// TIA Portal project "#06-J1500T(改角度）" (V17)

(* hardware
DEVICE "S7-1200 station_1"  S7-1200 Station
   slot 0: "Rack_0"  S7-1200 Rack  Rack  V1.0
   slot 1: "PLC_1"  CPU 1215C DC/DC/DC  6ES7 215-1AG40-0XB0  V4.5
   slot 2: "DI 16x24VDC_1"  6ES7 221-1BH32-0XB0  V2.0
   slot 3: "DI 16x24VDC_2"  6ES7 221-1BH32-0XB0  V2.0
   slot 4: "DI 16x24VDC_3"  6ES7 221-1BH32-0XB0  V2.0
   slot 5: "DQ 16x24VDC_1"  SM 1222 DQ16 x 24VDC  6ES7 222-1BH32-0XB0  V2.0
   slot 101: "CM 1243-5"  CM 1243-5  6GK7 243-5DX30-0XE0  V1.3
DEVICE "ET 200SP station_1"  ET 200SP-Station
   slot 0: "机架_0"  Rack  6ES5 710-8MAx1
   slot 0: "IO device_1"  IM 155-6 PN ST  6ES7 155-6AU01-0BN0  V4.2
   slot 1: "DI 16x24VDC ST_1"  DI 16x24VDC ST  6ES7 131-6BH01-0BA0  V0.0
      slot 1: "DI 16x24VDC ST_1"  DI 16x24VDC ST
   slot 2: "DI 16x24VDC ST_6"  DI 16x24VDC ST  6ES7 131-6BH01-0BA0  V0.0
      slot 1: "DI 16x24VDC ST_6"  DI 16x24VDC ST
   slot 3: "DI 16x24VDC ST_5"  DI 16x24VDC ST  6ES7 131-6BH01-0BA0  V0.0
      slot 1: "DI 16x24VDC ST_5"  DI 16x24VDC ST
   slot 4: "DI 16x24VDC ST_4"  DI 16x24VDC ST  6ES7 131-6BH01-0BA0  V0.0
      slot 1: "DI 16x24VDC ST_4"  DI 16x24VDC ST
   slot 5: "DI 16x24VDC ST_3"  DI 16x24VDC ST  6ES7 131-6BH01-0BA0  V0.0
      slot 1: "DI 16x24VDC ST_3"  DI 16x24VDC ST
   slot 6: "DQ 16x24VDC/0.5A ST_2"  DQ 16x24VDC/0.5A ST  6ES7 132-6BH01-0BA0  V0.0
      slot 1: "DQ 16x24VDC/0.5A ST_2"  DQ 16x24VDC/0.5A ST
   slot 7: "DQ 16x24VDC/0.5A ST_1"  DQ 16x24VDC/0.5A ST  6ES7 132-6BH01-0BA0  V0.0
      slot 1: "DQ 16x24VDC/0.5A ST_1"  DQ 16x24VDC/0.5A ST
   slot 8: "服务器模块_1"  Server module  6ES7 193-6PA00-0AA0  V1.1
      slot 1: "服务器模块_1"  Server module
   slot 127: "BA 2xRJ45"  BA 2xRJ45  6ES7 193-6AR00-0AA0  V0.0
      slot 1: "Port_1"  X1 P1 R  6ES7 193-6AR00-0AA0  V0.0
      slot 2: "Port_2"  X1 P2 R  6ES7 193-6AR00-0AA0  V0.0
DEVICE "HMI_1"  TP900 Comfort
   slot 0: "HMI_1"  TP900 Comfort  6AV2 124-0JC01-0AX0  15.1.0.0
   slot 1: "HMI_RT_1"  TP900 Comfort  6AV2 124-0JC01-0AX0  15.1.0.0
   slot 5: "HMI_1.IE_CP_1"  PROFINET Interface  15.0.1.0
      slot 1: "PROFINET Interface_1"  PROFINET Interface
         slot 1: "Port_1"  Port
         slot 2: "Port_2"  Port
   slot 7: "HMI_1.MPI/DP_CP_1"  MPI/DP Interface  15.0.1.0
DEVICE "GSD device_2"  GSD.Device
   slot 0: "机架_0"  Rail
   slot 0: "横梁站"  P+F  Encoder  4.0
DEVICE "GSD device_1"  GSD.Device
   slot 0: "机架_0"  Rail
   slot 0: "滑块站"  P+F  Encoder  4.0
*)

// ===== PLC "PLC_1"  CPU 1215C DC/DC/DC =====

VAR_GLOBAL   // PLC tag table "默认变量表"
   "Tag_1" AT %I0.0 : Bool;
   "Tag_136" AT %I19.3 : Bool;
   "Tag_137" AT %I19.4 : Bool;
   "Tag_138" AT %I19.5 : Bool;
   "Tag_139" AT %I19.6 : Bool;
   "Tag_140" AT %I19.7 : Bool;
   "机械凸轮单次返回" AT %I19.2 : Bool;
   "机械凸轮单次允许" AT %I19.1 : Bool;
   "机械凸轮上死点" AT %I19.0 : Bool;
   "右后双手闭点" AT %I18.7 : Bool;
   "Tag_46(1)" AT %I6.0 : Bool;
   "Tag_47(1)" AT %I6.1 : Bool;
   "Tag_48(1)" AT %I6.2 : Bool;
   "Tag_49(1)" AT %I6.3 : Bool;
   "Tag_50(1)" AT %I6.4 : Bool;
   "Tag_51(1)" AT %I6.5 : Bool;
   "Tag_52(1)" AT %I6.6 : Bool;
   "Tag_53(1)" AT %I6.7 : Bool;
   "Tag_54(1)" AT %I7.0 : Bool;
   "Tag_55(1)" AT %I7.1 : Bool;
   "Tag_56(1)" AT %I7.2 : Bool;
   "Tag_57(1)" AT %I7.3 : Bool;
   "Tag_58(1)" AT %I7.4 : Bool;
   "Tag_59" AT %I7.5 : Bool;
   "Tag_60" AT %I7.6 : Bool;
   "Tag_61(1)" AT %I7.7 : Bool;
   "工作台夹紧压检" AT %I18.0 : Bool;
   "工作台放松压检" AT %I18.1 : Bool;
   "故障复位" AT %I12.4 : Bool;
   "Tag_128" AT %I18.3 : Bool;
   "Tag_129" AT %I18.4 : Bool;
   "Tag_130" AT %I18.5 : Bool;
   "右后双手开点" AT %I18.6 : Bool;
   "Tag_108" AT %I15.7 : Bool;
   "平衡缸气压检测" AT %I15.6 : Bool;
   "Tag_105" AT %I15.4 : Bool;
   "Tag_28(1)" AT %I3.7 : Bool;
   "主电机启动接触器接通" AT %I3.5 : Bool;
   "Tag_26" AT %I3.4 : Bool;
   "Tag_25" AT %I3.3 : Bool;
   "Tag_2" AT %I0.1 : Bool;
   "Tag_3" AT %I0.2 : Bool;
   "Tag_4" AT %I0.3 : Bool;
   "Tag_5" AT %I0.4 : Bool;
   "Tag_6" AT %I0.5 : Bool;
   "Tag_7" AT %I0.6 : Bool;
   "Tag_8" AT %I0.7 : Bool;
   "Tag_9" AT %I1.0 : Bool;
   "Tag_10" AT %I1.1 : Bool;
   "Tag_11" AT %I1.2 : Bool;
   "Tag_12" AT %I1.3 : Bool;
   "Tag_13" AT %I1.4 : Bool;
   "Tag_14" AT %I1.5 : Bool;
   "Tag_15" AT %I2.1 : Bool;
   "Tag_16" AT %I2.2 : Bool;
   "Tag_17" AT %I2.3 : Bool;
   "KM17" AT %I2.4 : Bool;
   "Tag_19" AT %I2.5 : Bool;
   "Tag_20" AT %I2.6 : Bool;
   "Tag_21" AT %I2.7 : Bool;
   "KM12" AT %I3.0 : Bool;
   "Tag_23" AT %I3.1 : Bool;
   "KM11" AT %I3.2 : Bool;
   "Tag_35(1)" AT %I4.5 : Bool;
   "Tag_36(1)" AT %I4.6 : Bool;
   "Tag_37(1)" AT %I4.7 : Bool;
   "Tag_38(1)" AT %I5.0 : Bool;
   "Tag_39(1)" AT %I5.1 : Bool;
   "Tag_40(1)" AT %I5.2 : Bool;
   "Tag_41(1)" AT %I5.3 : Bool;
   "Tag_42(1)" AT %I5.4 : Bool;
   "Tag_43(1)" AT %I5.5 : Bool;
   "Tag_44(1)" AT %I5.6 : Bool;
   "Tag_45(1)" AT %I5.7 : Bool;
   "滑块调整选择" AT %I14.1 : Bool;
   "行程" AT %I14.2 : Bool;
   "气垫调整" AT %I14.3 : Bool;
   "模具更换" AT %I14.4 : Bool;
   "滑块向上" AT %I14.5 : Bool;
   "滑块向下" AT %I14.6 : Bool;
   "停上死点" AT %I14.7 : Bool;
   "Tag_101" AT %I15.0 : Bool;
   "滑块调整过扭矩" AT %I15.1 : Bool;
   "液压保护卸荷" AT %I15.2 : Bool;
   "液压保护压力检测" AT %I15.3 : Bool;
   "Tag_34(1)" AT %I4.4 : Bool;
   "爬梯开关" AT %I15.5 : Bool;
   "Tag_33(1)" AT %I4.3 : Bool;
   "Tag_31(1)" AT %I4.1 : Bool;
   "润滑停止按钮" AT %I10.0 : Bool;
   "润滑启动按钮" AT %I10.1 : Bool;
   "气垫手动润滑按钮" AT %I10.2 : Bool;
   "平衡缸手动润滑按钮" AT %I10.3 : Bool;
   "145" AT %I10.4 : Bool;
   "液压保护复位1" AT %I10.5 : Bool;
   "液压保护复位2" AT %I10.6 : Bool;
   "模具夹紧按钮" AT %I10.7 : Bool;
   "模具松开按钮" AT %I11.0 : Bool;
   "模具更换转换" AT %I11.1 : Bool;
   "工作台夹紧" AT %I11.2 : Bool;
   "工作台松开" AT %I11.3 : Bool;
   "微调启动按钮" AT %I11.4 : Bool;
   "微调正转" AT %I11.5 : Bool;
   "微调反转" AT %I11.6 : Bool;
   "主电机停止" AT %I11.7 : Bool;
   "Tag_30(1)" AT %I4.0 : Bool;
   "Tag_32(1)" AT %I4.2 : Bool;
   "Tag_61" AT %Q0.0 : Bool;
   "Tag_62" AT %Q0.1 : Bool;
   "Tag_63" AT %Q0.2 : Bool;
   "Tag_64" AT %Q0.3 : Bool;
   "Tag_65" AT %Q0.4 : Bool;
   "Tag_66" AT %Q0.5 : Bool;
   "Tag_68" AT %Q0.7 : Bool;
   "主电机正转DI1" AT %Q1.0 : Bool;
   "Tag_70" AT %Q1.1 : Bool;
   "润滑油泵启动2" AT %Q2.0 : Bool;
   "M6 ?" AT %Q2.1 : Bool;
   "KM3" AT %Q2.2 : Bool;
   "变频器上电" AT %Q2.3 : Bool;
   "气垫调整防粘连KM19" AT %Q2.4 : Bool;
   "气垫调整向上KM20" AT %Q2.5 : Bool;
   "气垫调整向下KM21" AT %Q2.6 : Bool;
   "Tag_67" AT %Q0.6 : Bool;
   "润滑油泵启动KM11" AT %Q2.7 : Bool;
   "滑块调整防粘连KM5" AT %Q3.0 : Bool;
   "滑块向上KM6" AT %Q3.1 : Bool;
   "滑块向下KM7" AT %Q3.2 : Bool;
   "制动器阀" AT %Q12.7 : Bool;
   "飞轮制动阀" AT %Q13.0 : Bool;
   "工作台夹紧阀(1)" AT %Q13.1 : Bool;
   "工作台放松阀(1)" AT %Q13.2 : Bool;
   "Tag_154" AT %Q13.3 : Bool;
   "Tag_155" AT %Q13.4 : Bool;
   "Tag_156" AT %Q13.5 : Bool;
   "Tag_157" AT %Q13.6 : Bool;
   "润滑指示灯" AT %Q13.7 : Bool;
   "下死点指示(1)" AT %Q10.0 : Bool;
   "离合器阀" AT %Q12.6 : Bool;
   "平衡缸润滑阀" AT %Q12.5 : Bool;
   "备用(4)" AT %Q12.3 : Bool;
   "KA41主电机正转" AT %Q3.3 : Bool;
   "Tag_83" AT %Q3.4 : Bool;
   "Tag_86" AT %Q3.5 : Bool;
   "Tag_87" AT %Q3.6 : Bool;
   "Tag_88" AT %Q3.7 : Bool;
   "上死点指示" AT %Q10.1 : Bool;
   "润滑油位低指示" AT %Q10.2 : Bool;
   "润滑油位高指示" AT %Q10.3 : Bool;
   "气垫润滑高压指示" AT %Q10.4 : Bool;
   "滤油器堵塞指示" AT %Q10.5 : Bool;
   "Tag_100" AT %Q10.6 : Bool;
   "Tag_102" AT %Q10.7 : Bool;
   "液压保护卸荷指示" AT %Q11.0 : Bool;
   "滑块调整过扭矩指示" AT %Q11.1 : Bool;
   "主电机运行指示" AT %Q11.2 : Bool;
   "连续预置指示" AT %Q11.3 : Bool;
   "Tag_109" AT %Q11.4 : Bool;
   "液压保护气源气阀(1)" AT %Q11.5 : Bool;
   "液压保护泵阀(1)" AT %Q11.6 : Bool;
   "Tag_142" AT %Q11.7 : Bool;
   "备用" AT %Q12.0 : Bool;
   "备用(1)" AT %Q12.1 : Bool;
   "备用(3)" AT %Q12.2 : Bool;
   "气垫润滑阀" AT %Q12.4 : Bool;
   "过滤器正常" AT %M5.0 : Bool;
   "润滑油压正常" AT %M5.1 : Bool;
   "滑块调整允许" AT %M5.2 : Bool;
   "急停故障" AT %M6.0 : Bool;
   "液压保护故障" AT %M6.1 : Bool;
   "气压故障" AT %M6.2 : Bool;
   "设备故障" AT %M6.3 : Bool;
   "滑块调整允许(1)" AT %M6.4 : Bool;
   "Tag_22" AT %MD20 : Time;
   "滑块调整允许2(1)" AT %M6.5 : Bool;
   "气垫调整允许" AT %M6.6 : Bool;
   "工作台移动允许" AT %M7.0 : Bool;
   "工作台落到位" AT %M7.1 : Bool;
   "润滑油泵启动OK" AT %M5.5 : Bool;
   "10度" AT %M200.0 : Bool;
   "20度" AT %M200.1 : Bool;
   "30度" AT %M200.2 : Bool;
   "40度" AT %M200.3 : Bool;
   "50" AT %M200.4 : Bool;
   "60" AT %M200.5 : Bool;
   "70" AT %M200.6 : Bool;
   "80" AT %M200.7 : Bool;
   "90" AT %M201.0 : Bool;
   "100" AT %M201.1 : Bool;
   "110" AT %M201.2 : Bool;
   "120" AT %M201.3 : Bool;
   "130" AT %M201.4 : Bool;
   "140" AT %M201.5 : Bool;
   "150" AT %M201.6 : Bool;
   "160" AT %M201.7 : Bool;
   "170" AT %M202.0 : Bool;
   "180" AT %M202.1 : Bool;
   "190" AT %M202.2 : Bool;
   "200" AT %M202.3 : Bool;
   "210" AT %M202.4 : Bool;
   "220" AT %M202.5 : Bool;
   "230" AT %M202.6 : Bool;
   "240" AT %M202.7 : Bool;
   "250" AT %M203.0 : Bool;
   "260" AT %M203.1 : Bool;
   "270" AT %M203.2 : Bool;
   "280" AT %M203.3 : Bool;
   "290" AT %M203.4 : Bool;
   "300" AT %M203.5 : Bool;
   "310" AT %M203.6 : Bool;
   "320" AT %M203.7 : Bool;
   "330" AT %M204.0 : Bool;
   "340" AT %M204.1 : Bool;
   "350" AT %M204.2 : Bool;
   "360" AT %M204.3 : Bool;
   "上死点" AT %M204.4 : Bool;
   "制动监控" AT %M204.5 : Bool;
   "下死点" AT %M204.6 : Bool;
   "单次返回" AT %M204.7 : Bool;
   "光电保护位置" AT %M205.0 : Bool;
   "横梁编码器" AT %ID68 : DWord;
   "滑块编码器" AT %ID72 : DInt;
   "主电机启动1" AT %I12.0 : Bool;
   "微调选择(1)" AT %I14.0 : Bool;
   "主电机启动2" AT %I12.1 : Bool;
   "寸动开点1" AT %I12.2 : Bool;
   "寸动闭点1" AT %I12.3 : Bool;
   "故障复位(1)" AT %I18.2 : Bool;
   "寸动开点2" AT %I12.5 : Bool;
   "寸动闭点2" AT %I12.6 : Bool;
   "Tag_34" AT %I12.7 : Bool;
   "Tag_35" AT %I13.0 : Bool;
   "选择连续" AT %I13.1 : Bool;
   "单次选择" AT %I13.2 : Bool;
   "选择寸动" AT %I13.3 : Bool;
   "Tag_39" AT %I13.4 : Bool;
   "急停闭点" AT %I13.5 : Bool;
   "急停开点1" AT %I13.6 : Bool;
   "急停开点2" AT %I13.7 : Bool;
   "润滑油位高" AT %I16.0 : Bool;
   "润滑油位低" AT %I16.1 : Bool;
   "Tag_45" AT %I16.2 : Bool;
   "润滑低压1" AT %I16.3 : Bool;
   "润滑低压2" AT %I16.4 : Bool;
   "润滑低压3" AT %I16.5 : Bool;
   "润滑高压" AT %I16.6 : Bool;
   "滤油器堵塞1" AT %I16.7 : Bool;
   "滤油器堵塞2" AT %I17.0 : Bool;
   "滤油器堵塞3" AT %I17.1 : Bool;
   "Tag_53" AT %I17.2 : Bool;
   "工作台落到位前" AT %I17.3 : Bool;
   "工作台落到位后" AT %I17.4 : Bool;
   "气垫落到位" AT %I17.5 : Bool;
   "右前双手开点" AT %I17.6 : Bool;
   "右前双手闭点" AT %I17.7 : Bool;
   "急停正常" AT %M10.0 : Bool;
   "行程允许" AT %M14.0 : Bool;
   "寸动允许" AT %M14.1 : Bool;
   "寸动开始" AT %M14.2 : Bool;
   "单次允许" AT %M14.3 : Bool;
   "单次开始" AT %M14.4 : Bool;
   "双手按钮开点" AT %M14.5 : Bool;
   "双手按钮闭点" AT %M14.6 : Bool;
   "编码器闭点监控" AT %M14.7 : Bool;
   "编码器开点监控" AT %M15.0 : Bool;
   "编码器故障" AT %M15.1 : Bool;
   "工作台-夹紧OK" AT %M15.2 : Bool;
   "工作台放松OK" AT %M15.3 : Bool;
   "润滑正常" AT %M15.4 : Bool;
   "滑块软限位上" AT %M15.5 : Bool;
   "滑块软限位下" AT %M15.6 : Bool;
   "上调整设定值" AT %M15.7 : Bool;
   "滑块调整自动向上" AT %M16.0 : Bool;
   "滑块调整自动向下" AT %M16.1 : Bool;
   "滑块调整自动选择" AT %M16.2 : Bool;
   "滑块手动调整" AT %M16.3 : Bool;
   "滑块调整手动/自动" AT %M301.5 : Bool;
   "ECamdata _DB_D{10}滑块设定高度" AT %MD150 : Real;
   "润滑检测时间" AT %M600.0 : Bool;
   "气垫向上调整" AT %M220.0 : Bool;
   "气垫向下调整" AT %M220.1 : Bool;
   "System_Byte" AT %MB1 : Byte;
   "FirstScan" AT %M1.0 : Bool;
   "DiagStatusUpdate" AT %M1.1 : Bool;
   "AlwaysTRUE" AT %M1.2 : Bool;
   "AlwaysFALSE" AT %M1.3 : Bool;
   "Clock_Byte" AT %MB0 : Byte;
   "Clock_10Hz" AT %M0.0 : Bool;
   "Clock_5Hz" AT %M0.1 : Bool;
   "Clock_2.5Hz" AT %M0.2 : Bool;
   "Clock_2Hz" AT %M0.3 : Bool;
   "Clock_1.25Hz" AT %M0.4 : Bool;
   "Clock_1Hz" AT %M0.5 : Bool;
   "Clock_0.625Hz" AT %M0.6 : Bool;
   "Clock_0.5Hz" AT %M0.7 : Bool;
   "主电机启动标志" AT %M700.0 : Bool;
   "爬梯占位" AT %M5000.1 : Bool;
   "正传选择（占位）" AT %M5000.2 : Bool;
   "反转选择（占位）" AT %M5000.3 : Bool;
   "正转启动标志" AT %M700.1 : Bool;
   "反转启动标志" AT %M700.2 : Bool;
   "主电机反转（占位）" AT %M5000.4 : Bool;
   "主电机转速稳定" AT %M700.3 : Bool;
   "横梁编码器通讯故障" AT %M700.5 : Bool;
   "滑块编码器通讯故障" AT %M700.6 : Bool;
   "ET200通讯故障" AT %M700.7 : Bool;
   "单次允许1" AT %M205.2 : Bool;
   "Tag_18" AT %M19.2 : Bool;
   "防重复角度" AT %M205.1 : Bool;
   "防重复监控" AT %M702.0 : Bool;
   "单次条件3" AT %M18.1 : Bool;
   "临时屏蔽" AT %M1000.0 : Bool;
END_VAR

VAR_GLOBAL   // PLC tag table "变量表"
   "平衡缸压力模拟量" AT %ID80 : DWord;
   "气垫压力模拟量" AT %ID81 : DWord;
   "Tag_108(1)" AT %QW570 : Int;
   "Tag_109(1)" AT %QW572 : Int;
   "报警1" AT %M3000.0 : Bool;
   "报警2" AT %M3000.1 : Bool;
   "报警3" AT %M3000.2 : Bool;
   "报警4" AT %M3000.3 : Bool;
   "报警5" AT %M3000.4 : Bool;
   "报警6" AT %M3000.5 : Bool;
   "报警7" AT %M3000.6 : Bool;
   "报警8" AT %M3000.7 : Bool;
   "报警9" AT %M3001.0 : Bool;
   "报警10" AT %M3001.1 : Bool;
   "报警11" AT %M3001.2 : Bool;
   "报警12" AT %M3001.3 : Bool;
   "报警13" AT %M3001.4 : Bool;
   "报警14" AT %M3001.5 : Bool;
   "报警15" AT %M3001.6 : Bool;
   "报警16" AT %M3001.7 : Bool;
   "PLC报警变量组1" AT %MW3000 : Int;
   "PLC报警变量组2" AT %MW3002 : Int;
   "PLC报警变量组3" AT %MW3004 : Int;
   "报警17" AT %M3002.0 : Bool;
   "报警18" AT %M3002.1 : Bool;
   "报警19" AT %M3002.2 : Bool;
   "报警20" AT %M3002.3 : Bool;
   "报警21" AT %M3002.4 : Bool;
   "报警22" AT %M3002.5 : Bool;
   "报警23" AT %M3002.6 : Bool;
   "报警24" AT %M3002.7 : Bool;
   "报警25" AT %M3003.0 : Bool;
   "报警26" AT %M3003.1 : Bool;
   "报警27" AT %M3003.2 : Bool;
   "报警28" AT %M3003.3 : Bool;
   "报警29" AT %M3003.4 : Bool;
   "报警30" AT %M3003.5 : Bool;
   "报警31" AT %M3003.6 : Bool;
   "报警32" AT %M3003.7 : Bool;
   "报警33" AT %M3004.0 : Bool;
   "报警34" AT %M3004.1 : Bool;
   "报警35" AT %M3004.2 : Bool;
   "报警36" AT %M3004.3 : Bool;
   "报警37" AT %M3004.4 : Bool;
   "报警38" AT %M3004.5 : Bool;
   "报警39" AT %M3004.6 : Bool;
   "报警40" AT %M3004.7 : Bool;
   "报警41" AT %M3005.0 : Bool;
   "报警42" AT %M3005.1 : Bool;
   "报警43" AT %M3005.2 : Bool;
   "报警44" AT %M3005.3 : Bool;
   "报警45" AT %M3005.4 : Bool;
   "报警46" AT %M3005.5 : Bool;
   "报警47" AT %M3005.6 : Bool;
   "报警48" AT %M3005.7 : Bool;
   "Tag_1(1)" AT %M100.0 : Bool;
   "Tag_7(2)" AT %M100.1 : Bool;
   "异常报警1" AT %M1008.3 : Bool;
   "异常报警2" AT %M1008.4 : Bool;
   "计数开始" AT %M30.0 : Bool;
   "计数清零" AT %M30.1 : Bool;
   "产量到达" AT %M30.2 : Bool;
END_VAR

VAR_GLOBAL CONSTANT   // PLC tag table "变量表"
   "无(1)" : Pip := 65535;
   "自动更新(1)" : Pip := 0;
   "PIP 1(1)" : Pip := 1;
   "PIP 2(1)" : Pip := 2;
   "PIP 3(1)" : Pip := 3;
   "PIP 4(1)" : Pip := 4;
   "PIP OB 伺服(1)" : Pip := 32768;
   "Local~MC(1)" : Hw_SubModule := 51;
   "Local~Common(1)" : Hw_SubModule := 50;
   "Local~Device(1)" : Hw_Device := 32;
   "Local~Configuration(1)" : Hw_SubModule := 33;
   "Local~Exec(1)" : Hw_SubModule := 52;
   "Local(1)" : Hw_SubModule := 49;
   "Local~PROFINET_接口_1(1)" : Hw_Interface := 64;
   "Local~PROFINET_接口_1~端口_1(1)" : Hw_Interface := 65;
   "Local~HSC_1(1)" : Hw_Hsc := 257;
   "Local~HSC_2(1)" : Hw_Hsc := 258;
   "Local~HSC_3(1)" : Hw_Hsc := 259;
   "Local~HSC_4(1)" : Hw_Hsc := 260;
   "Local~HSC_5(1)" : Hw_Hsc := 261;
   "Local~HSC_6(1)" : Hw_Hsc := 262;
   "Local~AI_2_1" : Hw_SubModule := 263;
   "Local~DI_14_DQ_10_1(1)" : Hw_SubModule := 264;
   "Local~Pulse_1(1)" : Hw_Pwm := 265;
   "Local~Pulse_2(1)" : Hw_Pwm := 266;
   "Local~Pulse_3(1)" : Hw_Pwm := 267;
   "Local~Pulse_4(1)" : Hw_Pwm := 268;
   "Local~CM_1243-5~DP_接口(1)" : Hw_Interface := 269;
   "Local~CM_1243-5(1)" : Hw_SubModule := 271;
   "Local~PROFINET_IO-System(1)" : Hw_IoSystem := 272;
   "Local~DP-Mastersystem(1)" : Hw_IoSystem := 273;
   "Local~DI_16x24VDC_1(1)" : Hw_SubModule := 291;
   "Local~DI_16x24VDC_2(1)" : Hw_SubModule := 292;
   "Local~DQ_16x24VDC_1(1)" : Hw_SubModule := 293;
   "立柱右前操作站~Head" : Hw_Interface := 288;
   "立柱右前操作站~DPSlave" : Hw_DpSlave := 286;
   "立柱右前操作站~DI_32x24VDC_1" : Hw_SubModule := 289;
   "立柱右前操作站~AI_8x12BIT_1" : Hw_SubModule := 294;
   "立柱右前操作站~DI_32x24VDC_2" : Hw_SubModule := 295;
   "立柱右前操作站~DI_32x24VDC_3" : Hw_SubModule := 296;
   "立柱右前操作站~DI_32x24VDC_4" : Hw_SubModule := 297;
   "立柱右前操作站~DO_32x24VDC_0_5A_2" : Hw_SubModule := 299;
   "立柱右前操作站~DO_16x24VDC_0_5A_1" : Hw_SubModule := 290;
   "立柱右前操作站~DI_16x24VDC_1" : Hw_SubModule := 274;
   "横梁站~Head(1)" : Hw_Interface := 280;
   "横梁站~DPSlave(1)" : Hw_DpSlave := 278;
   "横梁站~P+F_Version_2_1_Singleturn_1(1)" : Hw_SubModule := 281;
   "OB_Main(1)" : OB_PCYCLE := 1;
   "OB_Cyclic interrupt" : OB_Cyclic := 30;
   "OB_RackStationFailure" : OB_Any := 86;
   "OB_Startup" : OB_STARTUP := 100;
   "滑块站~Head(1)" : Hw_Interface := 277;
   "滑块站~DPSlave(1)" : Hw_DpSlave := 275;
   "滑块站~32_Bit_Class_2_+_Speed_2_1" : Hw_SubModule := 282;
   "滑块站~32_Bit_Class_2_+_Speed_2_2" : Hw_SubModule := 283;
END_VAR

TYPE "用户数据类型_1"
   STRUCT
      Element_1 : Bool;
   END_STRUCT;
END_TYPE

// folder: 4.1_Line_Operation

TYPE "Operation_Mode"
   STRUCT
      Auto : Bool;
      Auto_Sim : Bool;
      APC : Bool;
      ATC : Bool;
      Man : Bool;
      Setup : Bool;
      工作模式 : UInt;
      零件表 : UInt;
   END_STRUCT;
END_TYPE

TYPE "4.1_Line_Operation"
   STRUCT
      Mode_Act : "Operation_Mode";
      Mode_Seting : "Operation_Mode";
      Recipes_Operation : "HMI_Recipe";
      HMI : Array[1..10] of "HMI_State";
   END_STRUCT;
END_TYPE

TYPE "HMI_Recipe"
   STRUCT
      Recipe : Struct
         Clear : Bool;
         Load : Bool;
         Save : Bool;
         Edit_No : Int;
         Recipe_Edit_Auth : Bool;
         Recipe_Edit_Wizard : Int;
         Load_Active : Bool;
         Save_Active : Bool;
         ii : Int;
         Load_Timer : IEC_TIMER;
         Save_Timer : IEC_TIMER;
      END_STRUCT;
      RecipeExport : Struct
         Done : Bool;
         Busy : Bool;
         Error : Bool;
         Status : Word;
      END_STRUCT;
      RecipeImport : Struct
         Done : Bool;
         Busy : Bool;
         Error : Bool;
         Status : Word;
      END_STRUCT;
   END_STRUCT;
END_TYPE

TYPE "HMI_State"
   STRUCT
      Command : Struct
         Doub_Part_Dropped_Mem : Bool;
         Part_Dropped_Mem : Bool;
         Part_Picker_Mem : Bool;
         Part_Done_Mem : Bool;
         Optim_Auth : Bool;
         Part_No_Chg_Auth : Bool;
      END_STRUCT;
      State : Struct
         Doub_Part_Dropped_Mem_1 : Bool;
         Part_Dropped_Mem_1 : Bool;
         Part_Picker_Mem_1 : Bool;
         Part_Done_Mem_1 : Bool;
      END_STRUCT;
   END_STRUCT;
END_TYPE

// folder: (top level)

DATA_BLOCK "中继"   // DB1
{ S7_Optimized_Access := 'TRUE' }
VERSION : 0.1
   VAR
      计数开关 : Bool;
      计数清零开关 : Bool;
      产量到达 : Bool;
   END_VAR
BEGIN
END_DATA_BLOCK

DATA_BLOCK "横梁编码器 _DB"   // DB3
{ S7_Optimized_Access := 'TRUE' }
VERSION : 0.1
   VAR
      "0.0" : Struct
         "+0.0" : DWord;
         "+4.0" : DWord;
         "+8.0" : DWord;
         "+12.0" : DWord;
      END_STRUCT;
      横梁 : Int;
      滑块 : Int;
      滑块_1 : DWord;
      "+0.3" : Int;
      "+0.4" : Int;
      "+0.5" : Int;
      "角度校准值(原+0.6）" : Int;
      编码器角度 : Int;
      "+0.7" : Int;
   END_VAR
   VAR RETAIN
      "+0.8" : Int;
   END_VAR
   VAR
      "+0.9" : Int;
      "+0.10" : Int;
      "0.11" : Real;
      平衡器分油器检测 : Int;
      横梁分油器检测 : Int;
      滑块分油器检测 : Int;
      气垫分油器检测 : Int;
      "+0.15" : Int;
      "+0.16" : Int;
      "+0.17" : Int;
      "+0.18" : Int;
      "+0.19" : Int;
      "+0.20" : Int;
      "+0.21" : Int;
      "+0.22" : Int;
      "+0.23" : Int;
      "+0.24" : Int;
      "+0.25" : Int;
      "+0.26" : Int;
      "+0.27" : Int;
      "+0.28" : Int;
      "+0.29" : Int;
      "+0.30" : Int;
      平衡器打油次数 : Int;
      主分油器打油次数 : Int;
      滑块打油次数 : Int;
      气点垫打油次数 : Int;
      "+0.35" : Int;
      "+0.36" : Int;
      "+0.37" : Int;
      "+0.38" : Int;
      "+0.39" : Int;
      "+0.40" : Int;
      "+0.41" : Int;
      "+0.42" : Int;
      "+0.43" : Int;
      "+0.44" : Int;
      "+0.45" : Int;
      "+0.46" : Int;
      "+0.47" : Int;
      "+0.48" : Int;
   END_VAR
   VAR RETAIN
      AI : Array[0..10] of DInt;
      D : Array[0..10] of Real;
   END_VAR
   VAR
      AQD : Real;
      产量设定 : Int;
      D107 : Real;
   END_VAR
BEGIN
END_DATA_BLOCK

DATA_BLOCK "数据块_2"   // DB6
{ S7_Optimized_Access := 'TRUE' }
VERSION : 0.1
BEGIN
END_DATA_BLOCK

DATA_BLOCK "ECamdata _DB"   // DB7
{ S7_Optimized_Access := 'TRUE' }
VERSION : 0.1
   VAR
      "0.0" : Struct
         "+0.0" : DWord;
         "+4.0" : DWord;
         "+8.0" : DWord;
         "+12.0" : DWord;
      END_STRUCT;
      横梁编码器 : Int;
      滑块编码器 : DInt;
      气垫编码器1 : DWord;
      气垫编码器2 : DWord;
      平衡器压力显示_3 : Int;
      电子凸轮编码器 : Int;
      "+0.5" : Real;
      电子凸轮编码器显示 : Int;
      "+0.7" : DInt;
      "+0.8" : Int;
      "+0.9" : Real;
      "+0.10_1" : Int;
      "+0.11" : Int;
      "+0.12" : Int;
      "+0.13" : Int;
      "+0.10" : Int;
      平衡器分油器检测 : Int;
      横梁分油器检测 : Int;
      滑块分油器检测 : Int;
      气垫分油器检测 : Int;
      "+0.15" : Int;
      "+0.16" : Int;
      "+0.17" : Int;
      "+0.18" : Int;
      "+0.19" : Int;
      "+0.20" : Int;
      "+0.21" : Int;
      "+0.22" : Int;
      "+0.23" : Int;
      "+0.24" : Int;
      "+0.25" : Int;
      "+0.26" : Int;
      "+0.27" : Int;
      "+0.28" : Int;
      "+0.29" : Int;
      "+0.30" : Int;
      平衡器打油次数 : Int;
      主分油器打油次数 : Int;
      滑块打油次数 : Int;
      气点垫打油次数 : Int;
      "+0.35" : Int;
      "+0.36" : Int;
      平衡器压力显示_2 : Real;
      平衡器压力显示_1 : Real;
      "+0.39" : Int;
      "+0.40" : Real;
      "+0.41" : Real;
      气垫模拟量 : Int;
      气垫模拟量_1 : Real;
      气垫模拟量_2 : Real;
      "+0.45" : DInt;
      "+0.46" : Int;
      "+0.47" : Real;
      "+0.48" : Int;
   END_VAR
   VAR RETAIN
      AI : Array[0..10] of DInt;
      D : Array[0..20] of Real;
   END_VAR
   VAR
      平衡器压力显示 : Real;
      AQD2 : Real;
      气垫模拟量显示1 : Real;
      气垫模拟量显示2 : Real;
      平衡器设置压力 : Real;
      气垫1压力设置 : Real;
      气垫2压力设置 : Real;
      D100 : Real;
      D101 : Int;
      D102 : Int;
      D103 : Real;
      D104 : Real;
      D105 : Real;
      D106 : Real;
      D107 : Int;
      D108 : Real;
      D109 : Real;
   END_VAR
   VAR RETAIN
      设置产量 : Int;
      当前产量 : Int;
      滑块位置 : Int;
   END_VAR
   VAR
      气垫位置 : Int;
   END_VAR
   VAR RETAIN
      D200 : DInt;
      D201 : Int;
   END_VAR
   VAR
      滑块中间值1 : Real;
   END_VAR
BEGIN
END_DATA_BLOCK

DATA_BLOCK "诊断数据"   // DB20
{ S7_Optimized_Access := 'TRUE' }
VERSION : 0.1
   VAR
      "横梁编码器-state" : Array[0..127] of Bool;
      "横梁编码器-return" : Word;
      "滑块编码器-state" : Array[0..127] of Bool;
      "滑块编码器-return" : Word;
      "ET200-state" : Array[0..127] of Bool;
      "ET200-return" : Word;
   END_VAR
BEGIN
END_DATA_BLOCK

DATA_BLOCK "中间变量"   // DB100
{ S7_Optimized_Access := 'TRUE' }
VERSION : 0.1
   VAR
      当前产量 : Int;
      目标产量 : Int;
   END_VAR
BEGIN
END_DATA_BLOCK

DATA_BLOCK "counter"   // DB101
{ S7_Optimized_Access := 'TRUE' }
VERSION : 0.1
   VAR
      产量计数 : IEC_COUNTER;
   END_VAR
BEGIN
END_DATA_BLOCK

DATA_BLOCK "timer"   // DB200
{ S7_Optimized_Access := 'TRUE' }
VERSION : 0.1
   VAR
      主电机转速稳定延时 : IEC_TIMER;
      清零防误触延时 : IEC_TIMER;
   END_VAR
BEGIN
END_DATA_BLOCK

// folder: 04_HMI_Comand_Config

DATA_BLOCK "Line_OP"   // DB10
{ S7_Optimized_Access := 'TRUE' }
VERSION : 0.1
BEGIN
END_DATA_BLOCK

// folder: System blocks/Program resources

DATA_BLOCK "IEC_Timer_0_DB_3"   // DB2
{ S7_Optimized_Access := 'TRUE' }
AUTHOR : Simatic
FAMILY : IEC
NAME : IEC_TMR
VERSION : 1.0
// stored: InstanceOfName IEC_TIMER
"IEC_TIMER"
BEGIN
END_DATA_BLOCK

DATA_BLOCK "IEC_Timer_0_DB_1"   // DB4
{ S7_Optimized_Access := 'TRUE' }
AUTHOR : Simatic
FAMILY : IEC
NAME : IEC_TMR
VERSION : 1.0
// stored: InstanceOfName IEC_TIMER
"IEC_TIMER"
BEGIN
END_DATA_BLOCK

DATA_BLOCK "IEC_Timer_0_DB_2"   // DB5
{ S7_Optimized_Access := 'TRUE' }
AUTHOR : Simatic
FAMILY : IEC
NAME : IEC_TMR
VERSION : 1.0
// stored: InstanceOfName IEC_TIMER
"IEC_TIMER"
BEGIN
END_DATA_BLOCK

DATA_BLOCK "当前产量"   // DB8
{ S7_Optimized_Access := 'TRUE' }
AUTHOR : Simatic
FAMILY : IEC
NAME : CNTR
VERSION : 1.0
// stored: InstanceOfName IEC_COUNTER
"IEC_COUNTER"
BEGIN
END_DATA_BLOCK

// folder: (top level)

FUNCTION "工作台移动" : Void   // FC1, LAD
{ S7_Optimized_Access := 'TRUE' }
VERSION : 0.1
BEGIN

REGION Network 2
   // 000000000000000000000000000000000000.
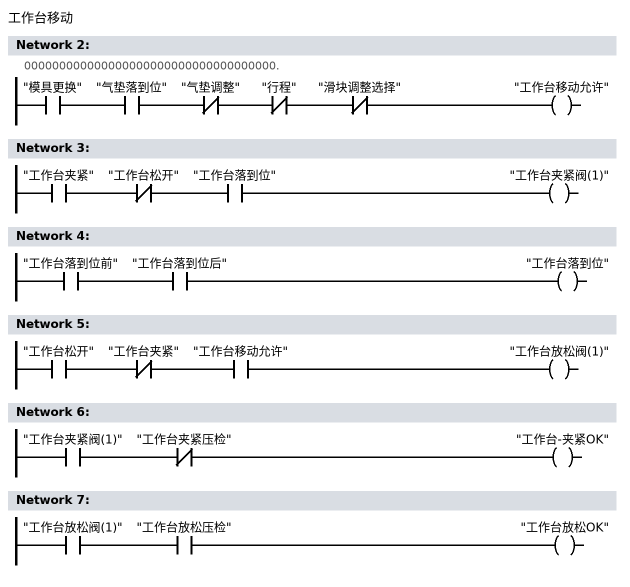
   RUNG wire#powerrail
      Contact( "模具更换" )
      Contact( "气垫落到位" )
      I_Contact( "气垫调整" )
      I_Contact( "行程" )
      I_Contact( "滑块调整选择" )
      Coil( "工作台移动允许" )
   END_RUNG
   // the same network as SCL:
   "工作台移动允许" := "模具更换" AND "气垫落到位" AND NOT "气垫调整" AND NOT "行程" AND NOT "滑块调整选择";
END_REGION

REGION Network 3
   RUNG wire#powerrail
      Contact( "工作台夹紧" )
      I_Contact( "工作台松开" )
      Contact( "工作台落到位" )
      Coil( "工作台夹紧阀(1)" )
   END_RUNG
   // the same network as SCL:
   "工作台夹紧阀(1)" := "工作台夹紧" AND NOT "工作台松开" AND "工作台落到位";
END_REGION

REGION Network 4
   RUNG wire#powerrail
      Contact( "工作台落到位前" )
      Contact( "工作台落到位后" )
      Coil( "工作台落到位" )
   END_RUNG
   // the same network as SCL:
   "工作台落到位" := "工作台落到位前" AND "工作台落到位后";
END_REGION

REGION Network 5
   RUNG wire#powerrail
      Contact( "工作台松开" )
      I_Contact( "工作台夹紧" )
      Contact( "工作台移动允许" )
      Coil( "工作台放松阀(1)" )
   END_RUNG
   // the same network as SCL:
   "工作台放松阀(1)" := "工作台松开" AND NOT "工作台夹紧" AND "工作台移动允许";
END_REGION

REGION Network 6
   RUNG wire#powerrail
      Contact( "工作台夹紧阀(1)" )
      I_Contact( "工作台夹紧压检" )
      Coil( "工作台-夹紧OK" )
   END_RUNG
   // the same network as SCL:
   "工作台-夹紧OK" := "工作台夹紧阀(1)" AND NOT "工作台夹紧压检";
END_REGION

REGION Network 7
   RUNG wire#powerrail
      Contact( "工作台放松阀(1)" )
      Contact( "工作台放松压检" )
      Coil( "工作台放松OK" )
   END_RUNG
   // the same network as SCL:
   "工作台放松OK" := "工作台放松阀(1)" AND "工作台放松压检";
END_REGION
END_FUNCTION

FUNCTION "横梁编码器调制" : Void   // FC2, LAD
{ S7_Optimized_Access := 'TRUE' }
VERSION : 0.1
BEGIN

REGION Network 1
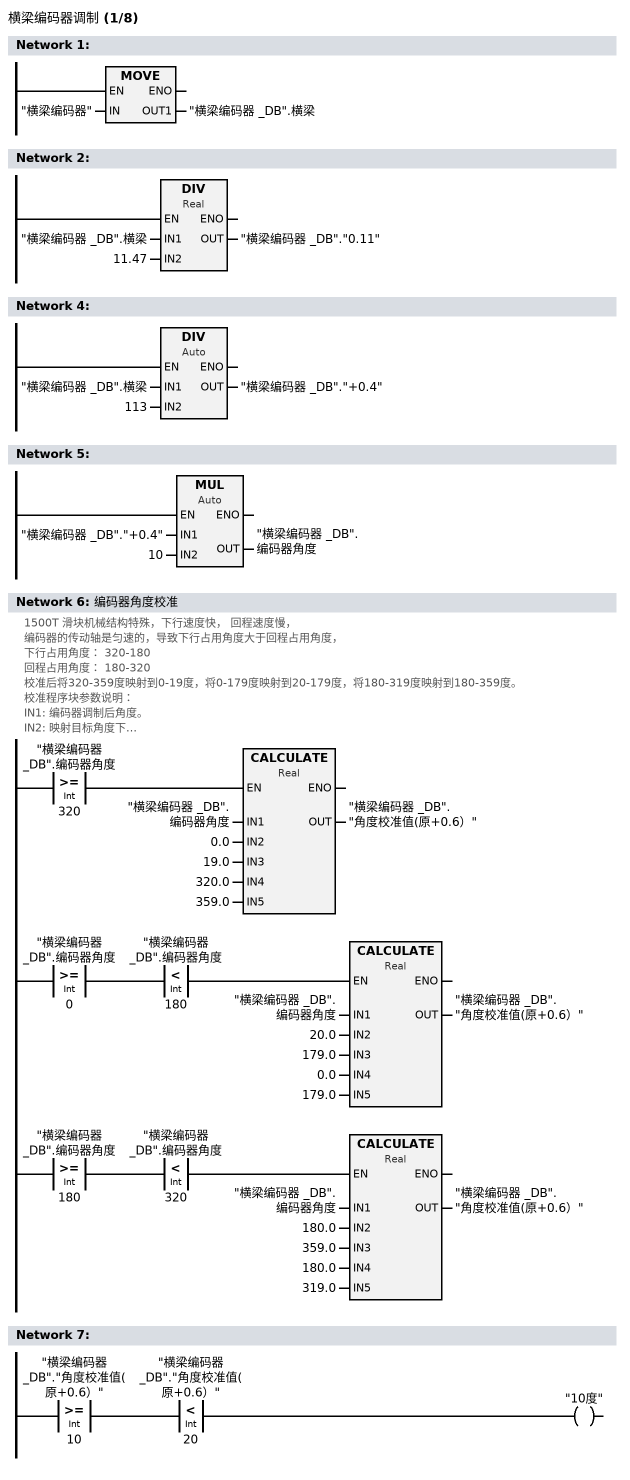
   RUNG wire#powerrail
      Move(in := "横梁编码器", out1 => "横梁编码器 _DB".横梁)
   END_RUNG
   // the same network as SCL:
   "横梁编码器 _DB".横梁 := "横梁编码器";
END_REGION

REGION Network 2
   RUNG wire#powerrail
      { S7_Templates := "SrcType := Real" } Div(in1 := "横梁编码器 _DB".横梁, in2 := 11.47, out => "横梁编码器 _DB"."0.11")
   END_RUNG
   // the same network as SCL:
   "横梁编码器 _DB"."0.11" := "横梁编码器 _DB".横梁 / 11.47;
END_REGION

REGION Network 4
   RUNG wire#powerrail
      Div(in1 := "横梁编码器 _DB".横梁, in2 := 113, out => "横梁编码器 _DB"."+0.4")
   END_RUNG
   // the same network as SCL:
   "横梁编码器 _DB"."+0.4" := "横梁编码器 _DB".横梁 / 113;
END_REGION

REGION Network 5
   RUNG wire#powerrail
      Mul(in1 := "横梁编码器 _DB"."+0.4", in2 := 10, out => "横梁编码器 _DB".编码器角度)
   END_RUNG
   // the same network as SCL:
   "横梁编码器 _DB".编码器角度 := "横梁编码器 _DB"."+0.4" * 10;
END_REGION

REGION Network 6: 编码器角度校准
   // 1500T 滑块机械结构特殊，下行速度快， 回程速度慢， 编码器的传动轴是匀速的，导致下行占用角度大于回程占用角度，
   // 下行占用角度： 320-180
   // 回程占用角度： 180-320
   // 校准后将320-359度映射到0-19度，将0-179度映射到20-179度，将180-319度映射到180-359度。 
   // 
   // 校准程序块参数说明： 
   // IN1: 编码器调制后角度。
   // IN2: 映射目标角度下限
   // IN3: 映射目标角度上限
   // IN4: 被映射角度下限
   // IN4: 被映射角度上限
   // OUT: 映射校准后的滑块实际角度
   RUNG wire#powerrail
      { S7_Templates := "SrcType := Int" } GE_Contact(in1 := "横梁编码器 _DB".编码器角度, in2 := 320)
      { S7_Templates := "SrcType := Real"; S7_Expression := "(IN1-IN4)/(IN5-IN4)*(IN3-IN2)+IN2" } Calculate(in1 := "横梁编码器 _DB".编码器角度, in2 := 0.0, in3 := 19.0, in4 := 320.0, in5 := 359.0, out => "横梁编码器 _DB"."角度校准值(原+0.6）")
   END_RUNG
   RUNG wire#powerrail
      { S7_Templates := "SrcType := Int" } GE_Contact(in1 := "横梁编码器 _DB".编码器角度, in2 := 0)
      { S7_Templates := "SrcType := Int" } LT_Contact(in1 := "横梁编码器 _DB".编码器角度, in2 := 180)
      { S7_Templates := "SrcType := Real"; S7_Expression := "(IN1-IN4)/(IN5-IN4)*(IN3-IN2)+IN2" } Calculate(in1 := "横梁编码器 _DB".编码器角度, in2 := 20.0, in3 := 179.0, in4 := 0.0, in5 := 179.0, out => "横梁编码器 _DB"."角度校准值(原+0.6）")
   END_RUNG
   RUNG wire#powerrail
      { S7_Templates := "SrcType := Int" } GE_Contact(in1 := "横梁编码器 _DB".编码器角度, in2 := 180)
      { S7_Templates := "SrcType := Int" } LT_Contact(in1 := "横梁编码器 _DB".编码器角度, in2 := 320)
      { S7_Templates := "SrcType := Real"; S7_Expression := "(IN1-IN4)/(IN5-IN4)*(IN3-IN2)+IN2" } Calculate(in1 := "横梁编码器 _DB".编码器角度, in2 := 180.0, in3 := 359.0, in4 := 180.0, in5 := 319.0, out => "横梁编码器 _DB"."角度校准值(原+0.6）")
   END_RUNG
   // the same network as SCL:
   IF "横梁编码器 _DB".编码器角度 >= 320 THEN
       "横梁编码器 _DB"."角度校准值(原+0.6）" := ("横梁编码器 _DB".编码器角度-320.0)/(359.0-320.0)*(19.0-0.0)+0.0;
   END_IF;
   IF ("横梁编码器 _DB".编码器角度 >= 0) AND ("横梁编码器 _DB".编码器角度 < 180) THEN
       "横梁编码器 _DB"."角度校准值(原+0.6）" := ("横梁编码器 _DB".编码器角度-0.0)/(179.0-0.0)*(179.0-20.0)+20.0;
   END_IF;
   IF ("横梁编码器 _DB".编码器角度 >= 180) AND ("横梁编码器 _DB".编码器角度 < 320) THEN
       "横梁编码器 _DB"."角度校准值(原+0.6）" := ("横梁编码器 _DB".编码器角度-180.0)/(319.0-180.0)*(359.0-180.0)+180.0;
   END_IF;
END_REGION

REGION Network 7
   RUNG wire#powerrail
      { S7_Templates := "SrcType := Int" } GE_Contact(in1 := "横梁编码器 _DB"."角度校准值(原+0.6）", in2 := 10)
      { S7_Templates := "SrcType := Int" } LT_Contact(in1 := "横梁编码器 _DB"."角度校准值(原+0.6）", in2 := 20)
      Coil( "10度" )
   END_RUNG
   // the same network as SCL:
   "10度" := ("横梁编码器 _DB"."角度校准值(原+0.6）" >= 10) AND ("横梁编码器 _DB"."角度校准值(原+0.6）" < 20);
END_REGION

REGION Network 8
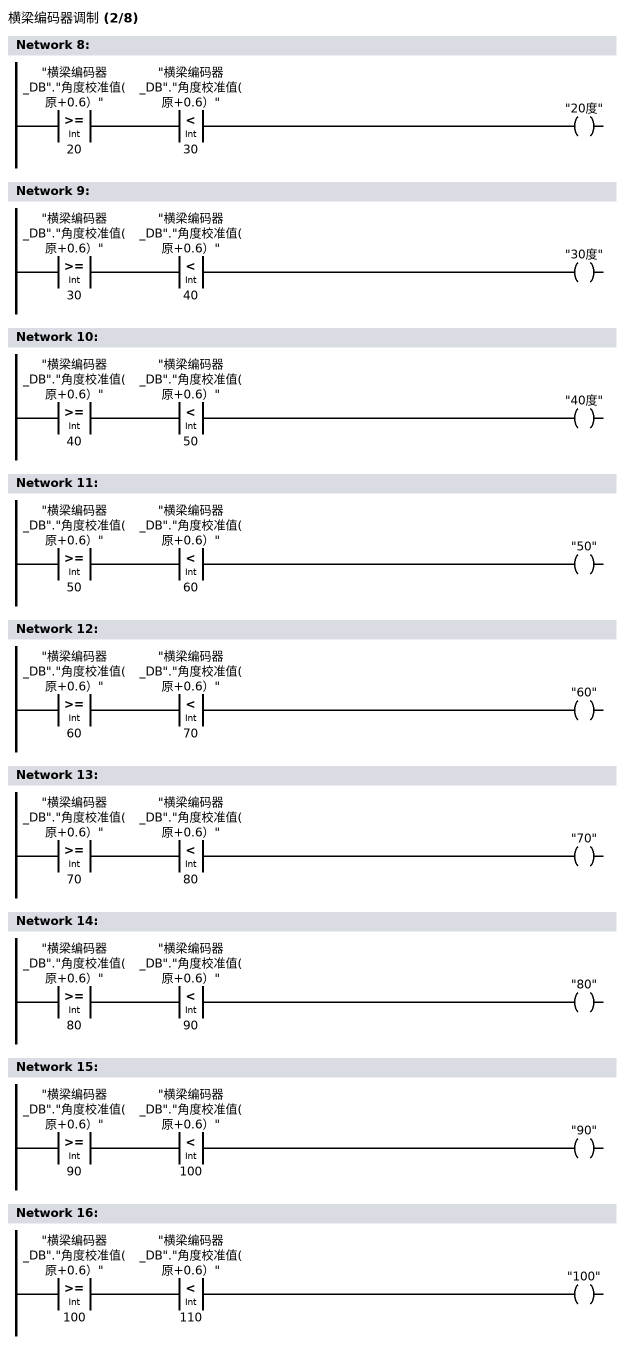
   RUNG wire#powerrail
      { S7_Templates := "SrcType := Int" } GE_Contact(in1 := "横梁编码器 _DB"."角度校准值(原+0.6）", in2 := 20)
      { S7_Templates := "SrcType := Int" } LT_Contact(in1 := "横梁编码器 _DB"."角度校准值(原+0.6）", in2 := 30)
      Coil( "20度" )
   END_RUNG
   // the same network as SCL:
   "20度" := ("横梁编码器 _DB"."角度校准值(原+0.6）" >= 20) AND ("横梁编码器 _DB"."角度校准值(原+0.6）" < 30);
END_REGION

REGION Network 9
   RUNG wire#powerrail
      { S7_Templates := "SrcType := Int" } GE_Contact(in1 := "横梁编码器 _DB"."角度校准值(原+0.6）", in2 := 30)
      { S7_Templates := "SrcType := Int" } LT_Contact(in1 := "横梁编码器 _DB"."角度校准值(原+0.6）", in2 := 40)
      Coil( "30度" )
   END_RUNG
   // the same network as SCL:
   "30度" := ("横梁编码器 _DB"."角度校准值(原+0.6）" >= 30) AND ("横梁编码器 _DB"."角度校准值(原+0.6）" < 40);
END_REGION

REGION Network 10
   RUNG wire#powerrail
      { S7_Templates := "SrcType := Int" } GE_Contact(in1 := "横梁编码器 _DB"."角度校准值(原+0.6）", in2 := 40)
      { S7_Templates := "SrcType := Int" } LT_Contact(in1 := "横梁编码器 _DB"."角度校准值(原+0.6）", in2 := 50)
      Coil( "40度" )
   END_RUNG
   // the same network as SCL:
   "40度" := ("横梁编码器 _DB"."角度校准值(原+0.6）" >= 40) AND ("横梁编码器 _DB"."角度校准值(原+0.6）" < 50);
END_REGION

REGION Network 11
   RUNG wire#powerrail
      { S7_Templates := "SrcType := Int" } GE_Contact(in1 := "横梁编码器 _DB"."角度校准值(原+0.6）", in2 := 50)
      { S7_Templates := "SrcType := Int" } LT_Contact(in1 := "横梁编码器 _DB"."角度校准值(原+0.6）", in2 := 60)
      Coil( "50" )
   END_RUNG
   // the same network as SCL:
   "50" := ("横梁编码器 _DB"."角度校准值(原+0.6）" >= 50) AND ("横梁编码器 _DB"."角度校准值(原+0.6）" < 60);
END_REGION

REGION Network 12
   RUNG wire#powerrail
      { S7_Templates := "SrcType := Int" } GE_Contact(in1 := "横梁编码器 _DB"."角度校准值(原+0.6）", in2 := 60)
      { S7_Templates := "SrcType := Int" } LT_Contact(in1 := "横梁编码器 _DB"."角度校准值(原+0.6）", in2 := 70)
      Coil( "60" )
   END_RUNG
   // the same network as SCL:
   "60" := ("横梁编码器 _DB"."角度校准值(原+0.6）" >= 60) AND ("横梁编码器 _DB"."角度校准值(原+0.6）" < 70);
END_REGION

REGION Network 13
   RUNG wire#powerrail
      { S7_Templates := "SrcType := Int" } GE_Contact(in1 := "横梁编码器 _DB"."角度校准值(原+0.6）", in2 := 70)
      { S7_Templates := "SrcType := Int" } LT_Contact(in1 := "横梁编码器 _DB"."角度校准值(原+0.6）", in2 := 80)
      Coil( "70" )
   END_RUNG
   // the same network as SCL:
   "70" := ("横梁编码器 _DB"."角度校准值(原+0.6）" >= 70) AND ("横梁编码器 _DB"."角度校准值(原+0.6）" < 80);
END_REGION

REGION Network 14
   RUNG wire#powerrail
      { S7_Templates := "SrcType := Int" } GE_Contact(in1 := "横梁编码器 _DB"."角度校准值(原+0.6）", in2 := 80)
      { S7_Templates := "SrcType := Int" } LT_Contact(in1 := "横梁编码器 _DB"."角度校准值(原+0.6）", in2 := 90)
      Coil( "80" )
   END_RUNG
   // the same network as SCL:
   "80" := ("横梁编码器 _DB"."角度校准值(原+0.6）" >= 80) AND ("横梁编码器 _DB"."角度校准值(原+0.6）" < 90);
END_REGION

REGION Network 15
   RUNG wire#powerrail
      { S7_Templates := "SrcType := Int" } GE_Contact(in1 := "横梁编码器 _DB"."角度校准值(原+0.6）", in2 := 90)
      { S7_Templates := "SrcType := Int" } LT_Contact(in1 := "横梁编码器 _DB"."角度校准值(原+0.6）", in2 := 100)
      Coil( "90" )
   END_RUNG
   // the same network as SCL:
   "90" := ("横梁编码器 _DB"."角度校准值(原+0.6）" >= 90) AND ("横梁编码器 _DB"."角度校准值(原+0.6）" < 100);
END_REGION

REGION Network 16
   RUNG wire#powerrail
      { S7_Templates := "SrcType := Int" } GE_Contact(in1 := "横梁编码器 _DB"."角度校准值(原+0.6）", in2 := 100)
      { S7_Templates := "SrcType := Int" } LT_Contact(in1 := "横梁编码器 _DB"."角度校准值(原+0.6）", in2 := 110)
      Coil( "100" )
   END_RUNG
   // the same network as SCL:
   "100" := ("横梁编码器 _DB"."角度校准值(原+0.6）" >= 100) AND ("横梁编码器 _DB"."角度校准值(原+0.6）" < 110);
END_REGION

REGION Network 17
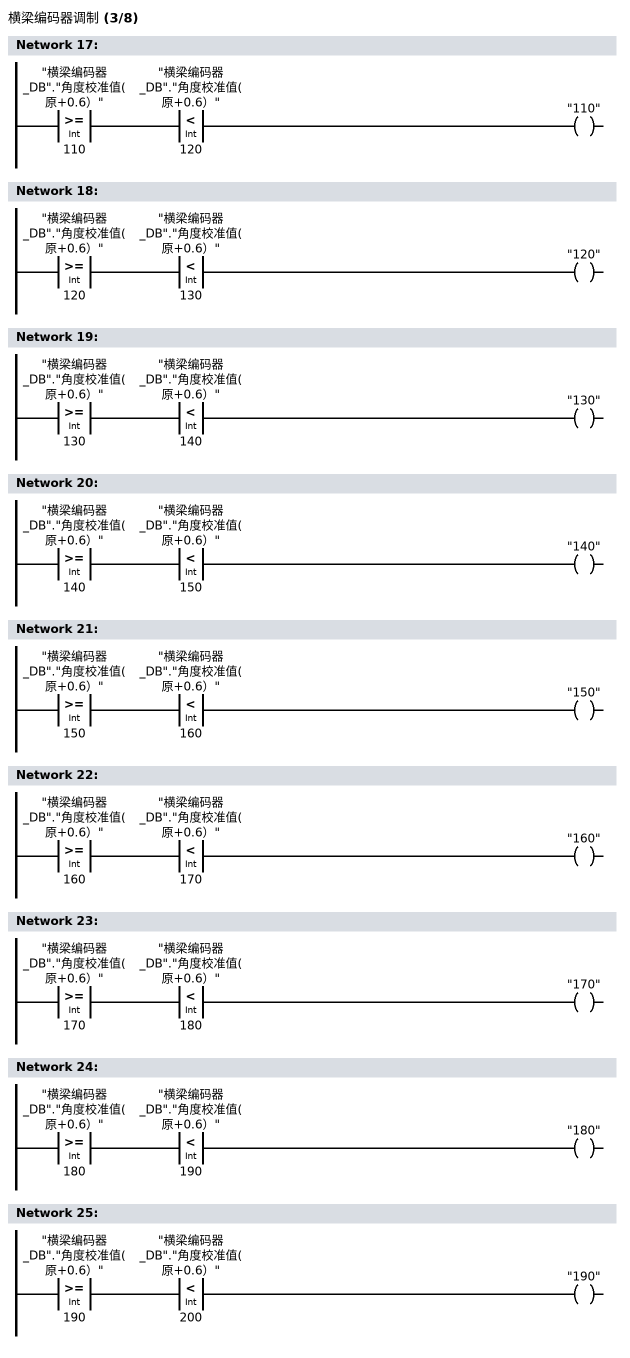
   RUNG wire#powerrail
      { S7_Templates := "SrcType := Int" } GE_Contact(in1 := "横梁编码器 _DB"."角度校准值(原+0.6）", in2 := 110)
      { S7_Templates := "SrcType := Int" } LT_Contact(in1 := "横梁编码器 _DB"."角度校准值(原+0.6）", in2 := 120)
      Coil( "110" )
   END_RUNG
   // the same network as SCL:
   "110" := ("横梁编码器 _DB"."角度校准值(原+0.6）" >= 110) AND ("横梁编码器 _DB"."角度校准值(原+0.6）" < 120);
END_REGION

REGION Network 18
   RUNG wire#powerrail
      { S7_Templates := "SrcType := Int" } GE_Contact(in1 := "横梁编码器 _DB"."角度校准值(原+0.6）", in2 := 120)
      { S7_Templates := "SrcType := Int" } LT_Contact(in1 := "横梁编码器 _DB"."角度校准值(原+0.6）", in2 := 130)
      Coil( "120" )
   END_RUNG
   // the same network as SCL:
   "120" := ("横梁编码器 _DB"."角度校准值(原+0.6）" >= 120) AND ("横梁编码器 _DB"."角度校准值(原+0.6）" < 130);
END_REGION

REGION Network 19
   RUNG wire#powerrail
      { S7_Templates := "SrcType := Int" } GE_Contact(in1 := "横梁编码器 _DB"."角度校准值(原+0.6）", in2 := 130)
      { S7_Templates := "SrcType := Int" } LT_Contact(in1 := "横梁编码器 _DB"."角度校准值(原+0.6）", in2 := 140)
      Coil( "130" )
   END_RUNG
   // the same network as SCL:
   "130" := ("横梁编码器 _DB"."角度校准值(原+0.6）" >= 130) AND ("横梁编码器 _DB"."角度校准值(原+0.6）" < 140);
END_REGION

REGION Network 20
   RUNG wire#powerrail
      { S7_Templates := "SrcType := Int" } GE_Contact(in1 := "横梁编码器 _DB"."角度校准值(原+0.6）", in2 := 140)
      { S7_Templates := "SrcType := Int" } LT_Contact(in1 := "横梁编码器 _DB"."角度校准值(原+0.6）", in2 := 150)
      Coil( "140" )
   END_RUNG
   // the same network as SCL:
   "140" := ("横梁编码器 _DB"."角度校准值(原+0.6）" >= 140) AND ("横梁编码器 _DB"."角度校准值(原+0.6）" < 150);
END_REGION

REGION Network 21
   RUNG wire#powerrail
      { S7_Templates := "SrcType := Int" } GE_Contact(in1 := "横梁编码器 _DB"."角度校准值(原+0.6）", in2 := 150)
      { S7_Templates := "SrcType := Int" } LT_Contact(in1 := "横梁编码器 _DB"."角度校准值(原+0.6）", in2 := 160)
      Coil( "150" )
   END_RUNG
   // the same network as SCL:
   "150" := ("横梁编码器 _DB"."角度校准值(原+0.6）" >= 150) AND ("横梁编码器 _DB"."角度校准值(原+0.6）" < 160);
END_REGION

REGION Network 22
   RUNG wire#powerrail
      { S7_Templates := "SrcType := Int" } GE_Contact(in1 := "横梁编码器 _DB"."角度校准值(原+0.6）", in2 := 160)
      { S7_Templates := "SrcType := Int" } LT_Contact(in1 := "横梁编码器 _DB"."角度校准值(原+0.6）", in2 := 170)
      Coil( "160" )
   END_RUNG
   // the same network as SCL:
   "160" := ("横梁编码器 _DB"."角度校准值(原+0.6）" >= 160) AND ("横梁编码器 _DB"."角度校准值(原+0.6）" < 170);
END_REGION

REGION Network 23
   RUNG wire#powerrail
      { S7_Templates := "SrcType := Int" } GE_Contact(in1 := "横梁编码器 _DB"."角度校准值(原+0.6）", in2 := 170)
      { S7_Templates := "SrcType := Int" } LT_Contact(in1 := "横梁编码器 _DB"."角度校准值(原+0.6）", in2 := 180)
      Coil( "170" )
   END_RUNG
   // the same network as SCL:
   "170" := ("横梁编码器 _DB"."角度校准值(原+0.6）" >= 170) AND ("横梁编码器 _DB"."角度校准值(原+0.6）" < 180);
END_REGION

REGION Network 24
   RUNG wire#powerrail
      { S7_Templates := "SrcType := Int" } GE_Contact(in1 := "横梁编码器 _DB"."角度校准值(原+0.6）", in2 := 180)
      { S7_Templates := "SrcType := Int" } LT_Contact(in1 := "横梁编码器 _DB"."角度校准值(原+0.6）", in2 := 190)
      Coil( "180" )
   END_RUNG
   // the same network as SCL:
   "180" := ("横梁编码器 _DB"."角度校准值(原+0.6）" >= 180) AND ("横梁编码器 _DB"."角度校准值(原+0.6）" < 190);
END_REGION

REGION Network 25
   RUNG wire#powerrail
      { S7_Templates := "SrcType := Int" } GE_Contact(in1 := "横梁编码器 _DB"."角度校准值(原+0.6）", in2 := 190)
      { S7_Templates := "SrcType := Int" } LT_Contact(in1 := "横梁编码器 _DB"."角度校准值(原+0.6）", in2 := 200)
      Coil( "190" )
   END_RUNG
   // the same network as SCL:
   "190" := ("横梁编码器 _DB"."角度校准值(原+0.6）" >= 190) AND ("横梁编码器 _DB"."角度校准值(原+0.6）" < 200);
END_REGION

REGION Network 26
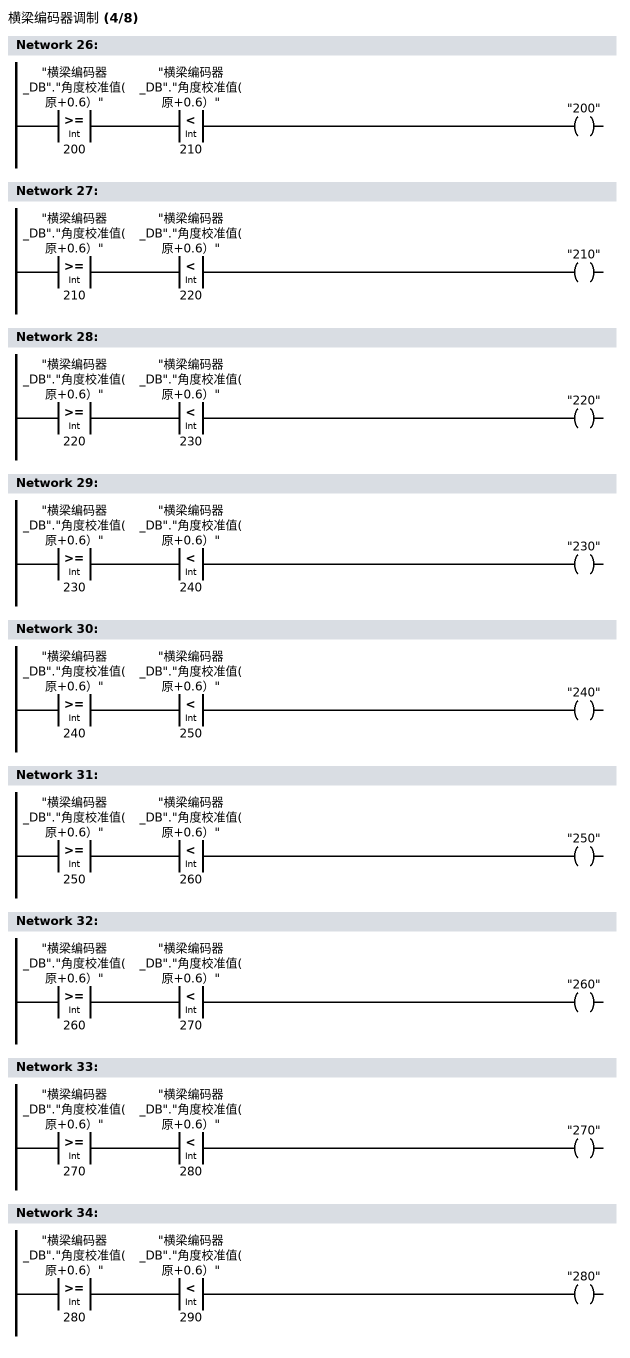
   RUNG wire#powerrail
      { S7_Templates := "SrcType := Int" } GE_Contact(in1 := "横梁编码器 _DB"."角度校准值(原+0.6）", in2 := 200)
      { S7_Templates := "SrcType := Int" } LT_Contact(in1 := "横梁编码器 _DB"."角度校准值(原+0.6）", in2 := 210)
      Coil( "200" )
   END_RUNG
   // the same network as SCL:
   "200" := ("横梁编码器 _DB"."角度校准值(原+0.6）" >= 200) AND ("横梁编码器 _DB"."角度校准值(原+0.6）" < 210);
END_REGION

REGION Network 27
   RUNG wire#powerrail
      { S7_Templates := "SrcType := Int" } GE_Contact(in1 := "横梁编码器 _DB"."角度校准值(原+0.6）", in2 := 210)
      { S7_Templates := "SrcType := Int" } LT_Contact(in1 := "横梁编码器 _DB"."角度校准值(原+0.6）", in2 := 220)
      Coil( "210" )
   END_RUNG
   // the same network as SCL:
   "210" := ("横梁编码器 _DB"."角度校准值(原+0.6）" >= 210) AND ("横梁编码器 _DB"."角度校准值(原+0.6）" < 220);
END_REGION

REGION Network 28
   RUNG wire#powerrail
      { S7_Templates := "SrcType := Int" } GE_Contact(in1 := "横梁编码器 _DB"."角度校准值(原+0.6）", in2 := 220)
      { S7_Templates := "SrcType := Int" } LT_Contact(in1 := "横梁编码器 _DB"."角度校准值(原+0.6）", in2 := 230)
      Coil( "220" )
   END_RUNG
   // the same network as SCL:
   "220" := ("横梁编码器 _DB"."角度校准值(原+0.6）" >= 220) AND ("横梁编码器 _DB"."角度校准值(原+0.6）" < 230);
END_REGION

REGION Network 29
   RUNG wire#powerrail
      { S7_Templates := "SrcType := Int" } GE_Contact(in1 := "横梁编码器 _DB"."角度校准值(原+0.6）", in2 := 230)
      { S7_Templates := "SrcType := Int" } LT_Contact(in1 := "横梁编码器 _DB"."角度校准值(原+0.6）", in2 := 240)
      Coil( "230" )
   END_RUNG
   // the same network as SCL:
   "230" := ("横梁编码器 _DB"."角度校准值(原+0.6）" >= 230) AND ("横梁编码器 _DB"."角度校准值(原+0.6）" < 240);
END_REGION

REGION Network 30
   RUNG wire#powerrail
      { S7_Templates := "SrcType := Int" } GE_Contact(in1 := "横梁编码器 _DB"."角度校准值(原+0.6）", in2 := 240)
      { S7_Templates := "SrcType := Int" } LT_Contact(in1 := "横梁编码器 _DB"."角度校准值(原+0.6）", in2 := 250)
      Coil( "240" )
   END_RUNG
   // the same network as SCL:
   "240" := ("横梁编码器 _DB"."角度校准值(原+0.6）" >= 240) AND ("横梁编码器 _DB"."角度校准值(原+0.6）" < 250);
END_REGION

REGION Network 31
   RUNG wire#powerrail
      { S7_Templates := "SrcType := Int" } GE_Contact(in1 := "横梁编码器 _DB"."角度校准值(原+0.6）", in2 := 250)
      { S7_Templates := "SrcType := Int" } LT_Contact(in1 := "横梁编码器 _DB"."角度校准值(原+0.6）", in2 := 260)
      Coil( "250" )
   END_RUNG
   // the same network as SCL:
   "250" := ("横梁编码器 _DB"."角度校准值(原+0.6）" >= 250) AND ("横梁编码器 _DB"."角度校准值(原+0.6）" < 260);
END_REGION

REGION Network 32
   RUNG wire#powerrail
      { S7_Templates := "SrcType := Int" } GE_Contact(in1 := "横梁编码器 _DB"."角度校准值(原+0.6）", in2 := 260)
      { S7_Templates := "SrcType := Int" } LT_Contact(in1 := "横梁编码器 _DB"."角度校准值(原+0.6）", in2 := 270)
      Coil( "260" )
   END_RUNG
   // the same network as SCL:
   "260" := ("横梁编码器 _DB"."角度校准值(原+0.6）" >= 260) AND ("横梁编码器 _DB"."角度校准值(原+0.6）" < 270);
END_REGION

REGION Network 33
   RUNG wire#powerrail
      { S7_Templates := "SrcType := Int" } GE_Contact(in1 := "横梁编码器 _DB"."角度校准值(原+0.6）", in2 := 270)
      { S7_Templates := "SrcType := Int" } LT_Contact(in1 := "横梁编码器 _DB"."角度校准值(原+0.6）", in2 := 280)
      Coil( "270" )
   END_RUNG
   // the same network as SCL:
   "270" := ("横梁编码器 _DB"."角度校准值(原+0.6）" >= 270) AND ("横梁编码器 _DB"."角度校准值(原+0.6）" < 280);
END_REGION

REGION Network 34
   RUNG wire#powerrail
      { S7_Templates := "SrcType := Int" } GE_Contact(in1 := "横梁编码器 _DB"."角度校准值(原+0.6）", in2 := 280)
      { S7_Templates := "SrcType := Int" } LT_Contact(in1 := "横梁编码器 _DB"."角度校准值(原+0.6）", in2 := 290)
      Coil( "280" )
   END_RUNG
   // the same network as SCL:
   "280" := ("横梁编码器 _DB"."角度校准值(原+0.6）" >= 280) AND ("横梁编码器 _DB"."角度校准值(原+0.6）" < 290);
END_REGION

REGION Network 35
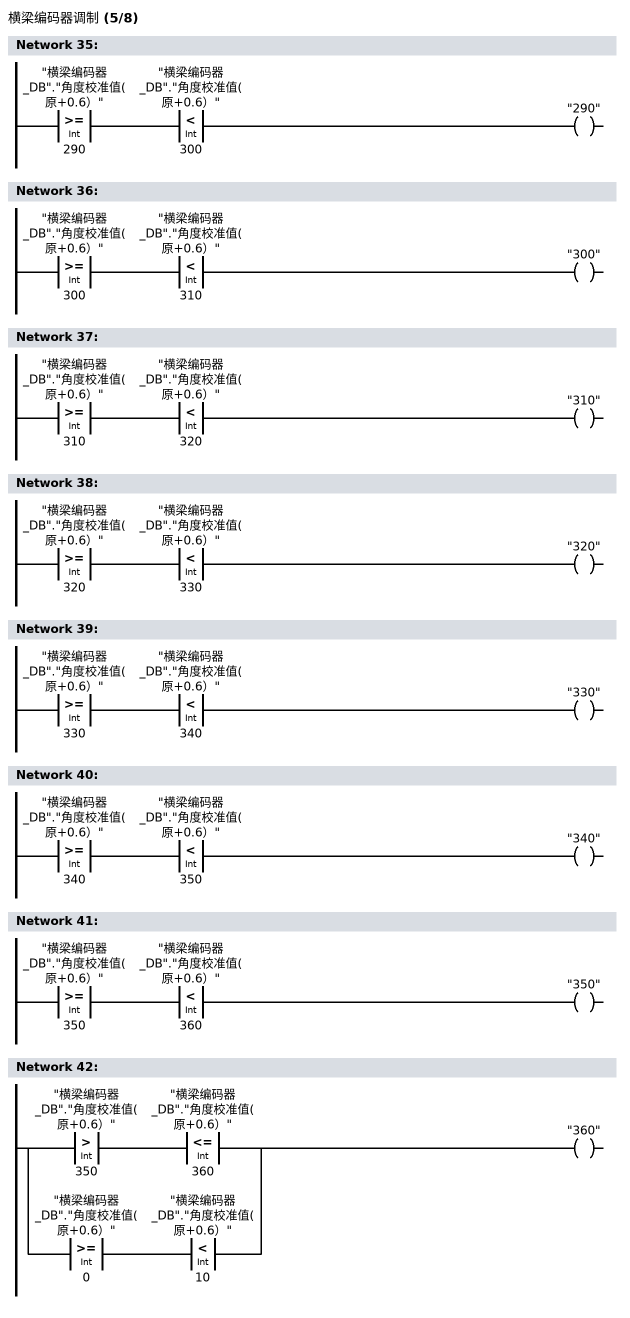
   RUNG wire#powerrail
      { S7_Templates := "SrcType := Int" } GE_Contact(in1 := "横梁编码器 _DB"."角度校准值(原+0.6）", in2 := 290)
      { S7_Templates := "SrcType := Int" } LT_Contact(in1 := "横梁编码器 _DB"."角度校准值(原+0.6）", in2 := 300)
      Coil( "290" )
   END_RUNG
   // the same network as SCL:
   "290" := ("横梁编码器 _DB"."角度校准值(原+0.6）" >= 290) AND ("横梁编码器 _DB"."角度校准值(原+0.6）" < 300);
END_REGION

REGION Network 36
   RUNG wire#powerrail
      { S7_Templates := "SrcType := Int" } GE_Contact(in1 := "横梁编码器 _DB"."角度校准值(原+0.6）", in2 := 300)
      { S7_Templates := "SrcType := Int" } LT_Contact(in1 := "横梁编码器 _DB"."角度校准值(原+0.6）", in2 := 310)
      Coil( "300" )
   END_RUNG
   // the same network as SCL:
   "300" := ("横梁编码器 _DB"."角度校准值(原+0.6）" >= 300) AND ("横梁编码器 _DB"."角度校准值(原+0.6）" < 310);
END_REGION

REGION Network 37
   RUNG wire#powerrail
      { S7_Templates := "SrcType := Int" } GE_Contact(in1 := "横梁编码器 _DB"."角度校准值(原+0.6）", in2 := 310)
      { S7_Templates := "SrcType := Int" } LT_Contact(in1 := "横梁编码器 _DB"."角度校准值(原+0.6）", in2 := 320)
      Coil( "310" )
   END_RUNG
   // the same network as SCL:
   "310" := ("横梁编码器 _DB"."角度校准值(原+0.6）" >= 310) AND ("横梁编码器 _DB"."角度校准值(原+0.6）" < 320);
END_REGION

REGION Network 38
   RUNG wire#powerrail
      { S7_Templates := "SrcType := Int" } GE_Contact(in1 := "横梁编码器 _DB"."角度校准值(原+0.6）", in2 := 320)
      { S7_Templates := "SrcType := Int" } LT_Contact(in1 := "横梁编码器 _DB"."角度校准值(原+0.6）", in2 := 330)
      Coil( "320" )
   END_RUNG
   // the same network as SCL:
   "320" := ("横梁编码器 _DB"."角度校准值(原+0.6）" >= 320) AND ("横梁编码器 _DB"."角度校准值(原+0.6）" < 330);
END_REGION

REGION Network 39
   RUNG wire#powerrail
      { S7_Templates := "SrcType := Int" } GE_Contact(in1 := "横梁编码器 _DB"."角度校准值(原+0.6）", in2 := 330)
      { S7_Templates := "SrcType := Int" } LT_Contact(in1 := "横梁编码器 _DB"."角度校准值(原+0.6）", in2 := 340)
      Coil( "330" )
   END_RUNG
   // the same network as SCL:
   "330" := ("横梁编码器 _DB"."角度校准值(原+0.6）" >= 330) AND ("横梁编码器 _DB"."角度校准值(原+0.6）" < 340);
END_REGION

REGION Network 40
   RUNG wire#powerrail
      { S7_Templates := "SrcType := Int" } GE_Contact(in1 := "横梁编码器 _DB"."角度校准值(原+0.6）", in2 := 340)
      { S7_Templates := "SrcType := Int" } LT_Contact(in1 := "横梁编码器 _DB"."角度校准值(原+0.6）", in2 := 350)
      Coil( "340" )
   END_RUNG
   // the same network as SCL:
   "340" := ("横梁编码器 _DB"."角度校准值(原+0.6）" >= 340) AND ("横梁编码器 _DB"."角度校准值(原+0.6）" < 350);
END_REGION

REGION Network 41
   RUNG wire#powerrail
      { S7_Templates := "SrcType := Int" } GE_Contact(in1 := "横梁编码器 _DB"."角度校准值(原+0.6）", in2 := 350)
      { S7_Templates := "SrcType := Int" } LT_Contact(in1 := "横梁编码器 _DB"."角度校准值(原+0.6）", in2 := 360)
      Coil( "350" )
   END_RUNG
   // the same network as SCL:
   "350" := ("横梁编码器 _DB"."角度校准值(原+0.6）" >= 350) AND ("横梁编码器 _DB"."角度校准值(原+0.6）" < 360);
END_REGION

REGION Network 42
   RUNG wire#powerrail
      { S7_Templates := "SrcType := Int" } GT_Contact(in1 := "横梁编码器 _DB"."角度校准值(原+0.6）", in2 := 350)
      { S7_Templates := "SrcType := Int" } LE_Contact(in1 := "横梁编码器 _DB"."角度校准值(原+0.6）", in2 := 360)
      wire#w1
      Coil( "360" )
   END_RUNG
   RUNG wire#powerrail
      { S7_Templates := "SrcType := Int" } GE_Contact(in1 := "横梁编码器 _DB"."角度校准值(原+0.6）", in2 := 0)
      { S7_Templates := "SrcType := Int" } LT_Contact(in1 := "横梁编码器 _DB"."角度校准值(原+0.6）", in2 := 10)
   END_RUNG wire#w1
   // the same network as SCL:
   "360" := (("横梁编码器 _DB"."角度校准值(原+0.6）" > 350) AND ("横梁编码器 _DB"."角度校准值(原+0.6）" <= 360)) OR (("横梁编码器 _DB"."角度校准值(原+0.6）" >= 0) AND ("横梁编码器 _DB"."角度校准值(原+0.6）" < 10));
END_REGION

REGION Network 43
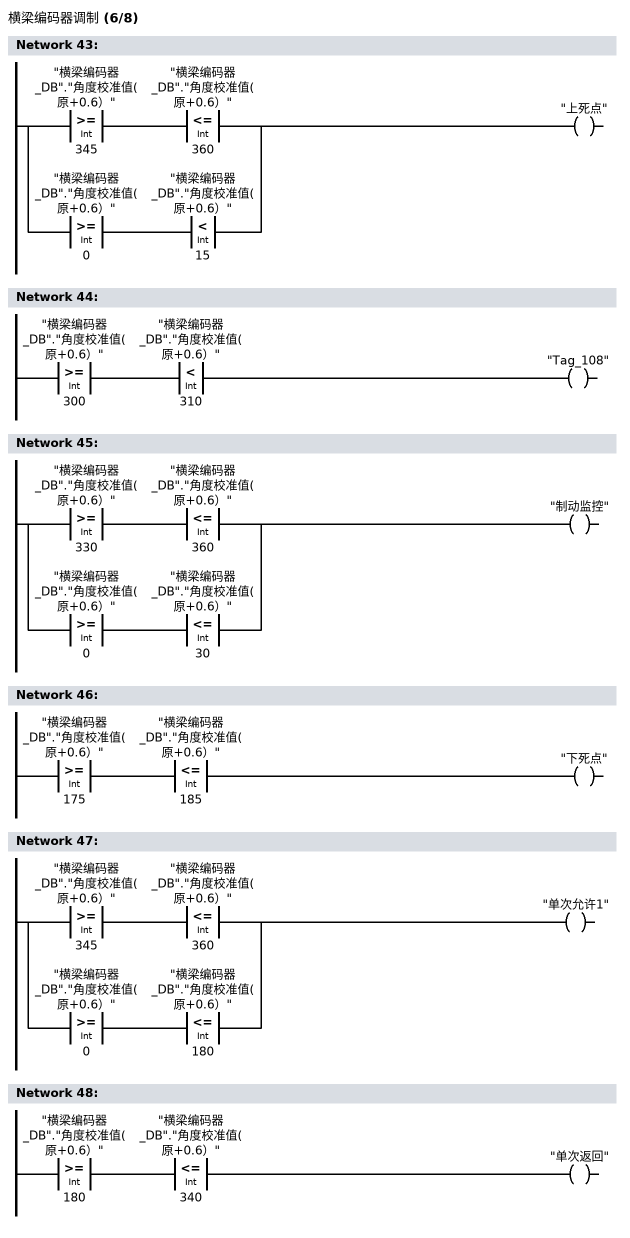
   RUNG wire#powerrail
      { S7_Templates := "SrcType := Int" } GE_Contact(in1 := "横梁编码器 _DB"."角度校准值(原+0.6）", in2 := 345)
      { S7_Templates := "SrcType := Int" } LE_Contact(in1 := "横梁编码器 _DB"."角度校准值(原+0.6）", in2 := 360)
      wire#w1
      Coil( "上死点" )
   END_RUNG
   RUNG wire#powerrail
      { S7_Templates := "SrcType := Int" } GE_Contact(in1 := "横梁编码器 _DB"."角度校准值(原+0.6）", in2 := 0)
      { S7_Templates := "SrcType := Int" } LT_Contact(in1 := "横梁编码器 _DB"."角度校准值(原+0.6）", in2 := 15)
   END_RUNG wire#w1
   // the same network as SCL:
   "上死点" := (("横梁编码器 _DB"."角度校准值(原+0.6）" >= 345) AND ("横梁编码器 _DB"."角度校准值(原+0.6）" <= 360)) OR (("横梁编码器 _DB"."角度校准值(原+0.6）" >= 0) AND ("横梁编码器 _DB"."角度校准值(原+0.6）" < 15));
END_REGION

REGION Network 44
   RUNG wire#powerrail
      { S7_Templates := "SrcType := Int" } GE_Contact(in1 := "横梁编码器 _DB"."角度校准值(原+0.6）", in2 := 300)
      { S7_Templates := "SrcType := Int" } LT_Contact(in1 := "横梁编码器 _DB"."角度校准值(原+0.6）", in2 := 310)
      Coil( "Tag_108" )
   END_RUNG
   // the same network as SCL:
   "Tag_108" := ("横梁编码器 _DB"."角度校准值(原+0.6）" >= 300) AND ("横梁编码器 _DB"."角度校准值(原+0.6）" < 310);
END_REGION

REGION Network 45
   RUNG wire#powerrail
      { S7_Templates := "SrcType := Int" } GE_Contact(in1 := "横梁编码器 _DB"."角度校准值(原+0.6）", in2 := 330)
      { S7_Templates := "SrcType := Int" } LE_Contact(in1 := "横梁编码器 _DB"."角度校准值(原+0.6）", in2 := 360)
      wire#w1
      Coil( "制动监控" )
   END_RUNG
   RUNG wire#powerrail
      { S7_Templates := "SrcType := Int" } GE_Contact(in1 := "横梁编码器 _DB"."角度校准值(原+0.6）", in2 := 0)
      { S7_Templates := "SrcType := Int" } LE_Contact(in1 := "横梁编码器 _DB"."角度校准值(原+0.6）", in2 := 30)
   END_RUNG wire#w1
   // the same network as SCL:
   "制动监控" := (("横梁编码器 _DB"."角度校准值(原+0.6）" >= 330) AND ("横梁编码器 _DB"."角度校准值(原+0.6）" <= 360)) OR (("横梁编码器 _DB"."角度校准值(原+0.6）" >= 0) AND ("横梁编码器 _DB"."角度校准值(原+0.6）" <= 30));
END_REGION

REGION Network 46
   RUNG wire#powerrail
      { S7_Templates := "SrcType := Int" } GE_Contact(in1 := "横梁编码器 _DB"."角度校准值(原+0.6）", in2 := 175)
      { S7_Templates := "SrcType := Int" } LE_Contact(in1 := "横梁编码器 _DB"."角度校准值(原+0.6）", in2 := 185)
      Coil( "下死点" )
   END_RUNG
   // the same network as SCL:
   "下死点" := ("横梁编码器 _DB"."角度校准值(原+0.6）" >= 175) AND ("横梁编码器 _DB"."角度校准值(原+0.6）" <= 185);
END_REGION

REGION Network 47
   RUNG wire#powerrail
      { S7_Templates := "SrcType := Int" } GE_Contact(in1 := "横梁编码器 _DB"."角度校准值(原+0.6）", in2 := 345)
      { S7_Templates := "SrcType := Int" } LE_Contact(in1 := "横梁编码器 _DB"."角度校准值(原+0.6）", in2 := 360)
      wire#w1
      Coil( "单次允许1" )
   END_RUNG
   RUNG wire#powerrail
      { S7_Templates := "SrcType := Int" } GE_Contact(in1 := "横梁编码器 _DB"."角度校准值(原+0.6）", in2 := 0)
      { S7_Templates := "SrcType := Int" } LE_Contact(in1 := "横梁编码器 _DB"."角度校准值(原+0.6）", in2 := 180)
   END_RUNG wire#w1
   // the same network as SCL:
   "单次允许1" := (("横梁编码器 _DB"."角度校准值(原+0.6）" >= 345) AND ("横梁编码器 _DB"."角度校准值(原+0.6）" <= 360)) OR (("横梁编码器 _DB"."角度校准值(原+0.6）" >= 0) AND ("横梁编码器 _DB"."角度校准值(原+0.6）" <= 180));
END_REGION

REGION Network 48
   RUNG wire#powerrail
      { S7_Templates := "SrcType := Int" } GE_Contact(in1 := "横梁编码器 _DB"."角度校准值(原+0.6）", in2 := 180)
      { S7_Templates := "SrcType := Int" } LE_Contact(in1 := "横梁编码器 _DB"."角度校准值(原+0.6）", in2 := 340)
      Coil( "单次返回" )
   END_RUNG
   // the same network as SCL:
   "单次返回" := ("横梁编码器 _DB"."角度校准值(原+0.6）" >= 180) AND ("横梁编码器 _DB"."角度校准值(原+0.6）" <= 340);
END_REGION

REGION Network 49
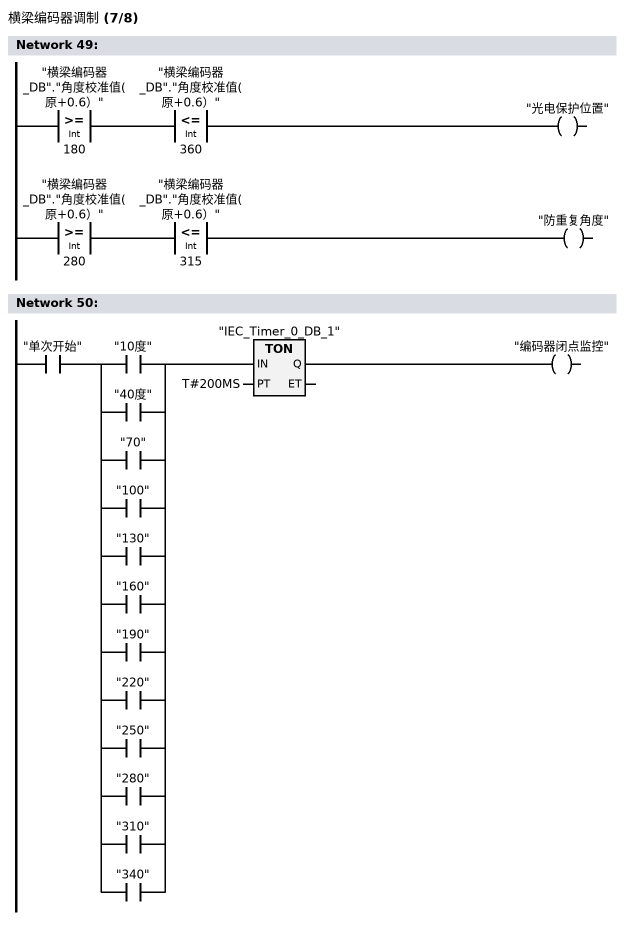
   RUNG wire#powerrail
      { S7_Templates := "SrcType := Int" } GE_Contact(in1 := "横梁编码器 _DB"."角度校准值(原+0.6）", in2 := 180)
      { S7_Templates := "SrcType := Int" } LE_Contact(in1 := "横梁编码器 _DB"."角度校准值(原+0.6）", in2 := 360)
      Coil( "光电保护位置" )
   END_RUNG
   RUNG wire#powerrail
      { S7_Templates := "SrcType := Int" } GE_Contact(in1 := "横梁编码器 _DB"."角度校准值(原+0.6）", in2 := 280)
      { S7_Templates := "SrcType := Int" } LE_Contact(in1 := "横梁编码器 _DB"."角度校准值(原+0.6）", in2 := 315)
      Coil( "防重复角度" )
   END_RUNG
   // the same network as SCL:
   "光电保护位置" := ("横梁编码器 _DB"."角度校准值(原+0.6）" >= 180) AND ("横梁编码器 _DB"."角度校准值(原+0.6）" <= 360);
   "防重复角度" := ("横梁编码器 _DB"."角度校准值(原+0.6）" >= 280) AND ("横梁编码器 _DB"."角度校准值(原+0.6）" <= 315);
END_REGION

REGION Network 50
   "IEC_Timer_0_DB_1".TON(IN := "单次开始" AND ("10度" OR "40度" OR "70" OR "100" OR "130" OR "160" OR "190" OR "220" OR "250" OR "280" OR "310" OR "340"),
                          PT := T#200MS);
   "编码器闭点监控" := "IEC_Timer_0_DB_1".Q;
END_REGION

REGION Network 51
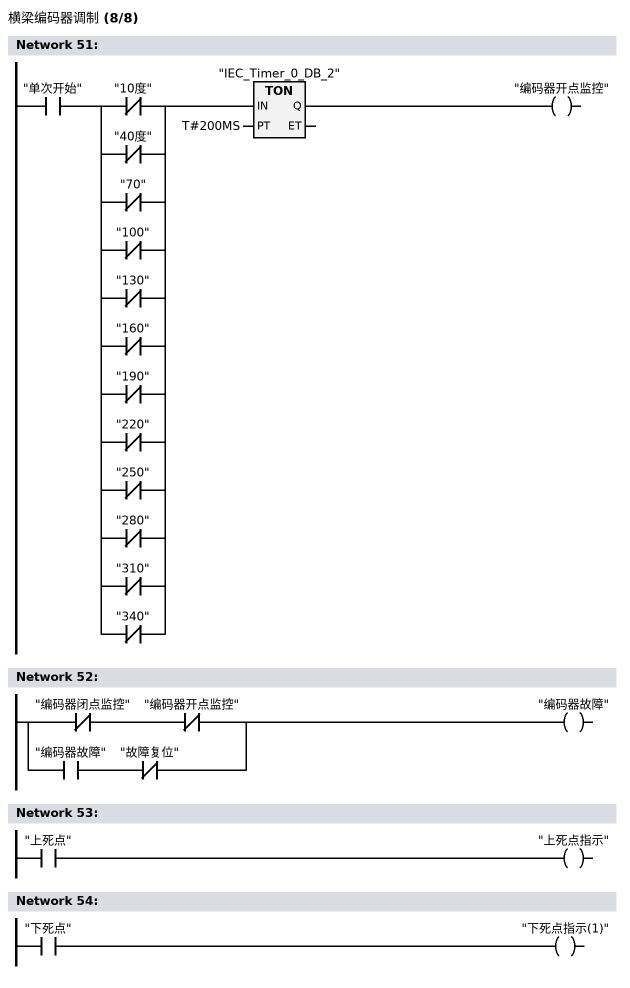
   "IEC_Timer_0_DB_2".TON(IN := "单次开始" AND (NOT "10度" OR NOT "40度" OR NOT "70" OR NOT "100" OR NOT "130" OR NOT "160" OR NOT "190" OR NOT "220" OR NOT "250" OR NOT "280" OR NOT "310" OR NOT "340"),
                          PT := T#200MS);
   "编码器开点监控" := "IEC_Timer_0_DB_2".Q;
END_REGION

REGION Network 52
   RUNG wire#powerrail
      I_Contact( "编码器闭点监控" )
      I_Contact( "编码器开点监控" )
      wire#w1
      Coil( "编码器故障" )
   END_RUNG
   RUNG wire#powerrail
      Contact( "编码器故障" )
      I_Contact( "故障复位" )
   END_RUNG wire#w1
   // the same network as SCL:
   "编码器故障" := (NOT "编码器闭点监控" AND NOT "编码器开点监控") OR ("编码器故障" AND NOT "故障复位");
END_REGION

REGION Network 53
   RUNG wire#powerrail
      Contact( "上死点" )
      Coil( "上死点指示" )
   END_RUNG
   // the same network as SCL:
   "上死点指示" := "上死点";
END_REGION

REGION Network 54
   RUNG wire#powerrail
      Contact( "下死点" )
      Coil( "下死点指示(1)" )
   END_RUNG
   // the same network as SCL:
   "下死点指示(1)" := "下死点";
END_REGION
END_FUNCTION

FUNCTION "滑块调整" : Void   // FC3, LAD
{ S7_Optimized_Access := 'TRUE' }
VERSION : 0.1
BEGIN

REGION Network 1
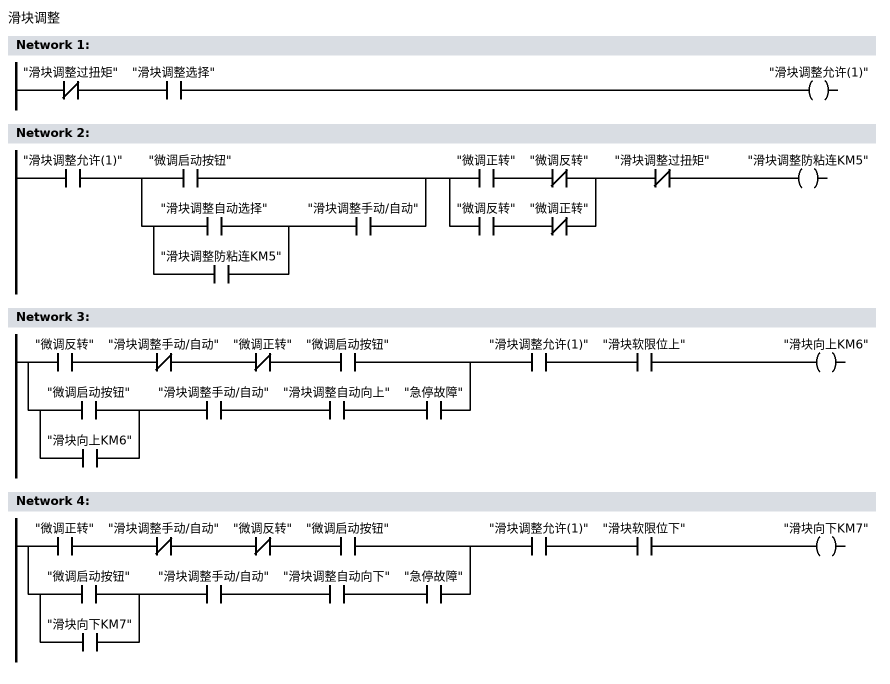
   RUNG wire#powerrail
      I_Contact( "滑块调整过扭矩" )
      Contact( "滑块调整选择" )
      Coil( "滑块调整允许(1)" )
   END_RUNG
   // the same network as SCL:
   "滑块调整允许(1)" := NOT "滑块调整过扭矩" AND "滑块调整选择";
END_REGION

REGION Network 2
   RUNG wire#powerrail
      Contact( "滑块调整允许(1)" )
      wire#w1
      Contact( "微调启动按钮" )
      wire#w2
      Contact( "微调正转" )
      I_Contact( "微调反转" )
      wire#w4
      I_Contact( "滑块调整过扭矩" )
      Coil( "滑块调整防粘连KM5" )
   END_RUNG
   RUNG wire#w1
      Contact( "滑块调整自动选择" )
      wire#w3
      Contact( "滑块调整手动/自动" )
   END_RUNG wire#w2
   RUNG wire#w1
      Contact( "滑块调整防粘连KM5" )
   END_RUNG wire#w3
   RUNG wire#w2
      Contact( "微调反转" )
      I_Contact( "微调正转" )
   END_RUNG wire#w4
   // the same network as SCL:
   "滑块调整防粘连KM5" := "滑块调整允许(1)" AND ("微调启动按钮" OR (("滑块调整自动选择" OR "滑块调整防粘连KM5") AND "滑块调整手动/自动")) AND (("微调正转" AND NOT "微调反转") OR ("微调反转" AND NOT "微调正转")) AND NOT "滑块调整过扭矩";
END_REGION

REGION Network 3
   RUNG wire#powerrail
      Contact( "微调反转" )
      I_Contact( "滑块调整手动/自动" )
      I_Contact( "微调正转" )
      Contact( "微调启动按钮" )
      wire#w1
      Contact( "滑块调整允许(1)" )
      Contact( "滑块软限位上" )
      Coil( "滑块向上KM6" )
   END_RUNG
   RUNG wire#powerrail
      Contact( "微调启动按钮" )
      wire#w2
      Contact( "滑块调整手动/自动" )
      Contact( "滑块调整自动向上" )
      Contact( "急停故障" )
   END_RUNG wire#w1
   RUNG wire#powerrail
      Contact( "滑块向上KM6" )
   END_RUNG wire#w2
   // the same network as SCL:
   "滑块向上KM6" := (("微调反转" AND NOT "滑块调整手动/自动" AND NOT "微调正转" AND "微调启动按钮") OR (("微调启动按钮" OR "滑块向上KM6") AND "滑块调整手动/自动" AND "滑块调整自动向上" AND "急停故障")) AND "滑块调整允许(1)" AND "滑块软限位上";
END_REGION

REGION Network 4
   RUNG wire#powerrail
      Contact( "微调正转" )
      I_Contact( "滑块调整手动/自动" )
      I_Contact( "微调反转" )
      Contact( "微调启动按钮" )
      wire#w1
      Contact( "滑块调整允许(1)" )
      Contact( "滑块软限位下" )
      Coil( "滑块向下KM7" )
   END_RUNG
   RUNG wire#powerrail
      Contact( "微调启动按钮" )
      wire#w2
      Contact( "滑块调整手动/自动" )
      Contact( "滑块调整自动向下" )
      Contact( "急停故障" )
   END_RUNG wire#w1
   RUNG wire#powerrail
      Contact( "滑块向下KM7" )
   END_RUNG wire#w2
   // the same network as SCL:
   "滑块向下KM7" := (("微调正转" AND NOT "滑块调整手动/自动" AND NOT "微调反转" AND "微调启动按钮") OR (("微调启动按钮" OR "滑块向下KM7") AND "滑块调整手动/自动" AND "滑块调整自动向下" AND "急停故障")) AND "滑块调整允许(1)" AND "滑块软限位下";
END_REGION
END_FUNCTION

FUNCTION "急停" : Void   // FC4, LAD
{ S7_Optimized_Access := 'TRUE' }
VERSION : 0.1
BEGIN

REGION Network 1
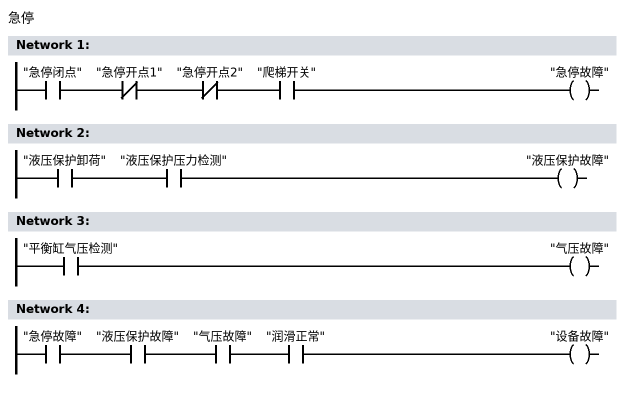
   RUNG wire#powerrail
      Contact( "急停闭点" )
      I_Contact( "急停开点1" )
      I_Contact( "急停开点2" )
      Contact( "爬梯开关" )
      Coil( "急停故障" )
   END_RUNG
   // the same network as SCL:
   "急停故障" := "急停闭点" AND NOT "急停开点1" AND NOT "急停开点2" AND "爬梯开关";
END_REGION

REGION Network 2
   RUNG wire#powerrail
      Contact( "液压保护卸荷" )
      Contact( "液压保护压力检测" )
      Coil( "液压保护故障" )
   END_RUNG
   // the same network as SCL:
   "液压保护故障" := "液压保护卸荷" AND "液压保护压力检测";
END_REGION

REGION Network 3
   RUNG wire#powerrail
      Contact( "平衡缸气压检测" )
      Coil( "气压故障" )
   END_RUNG
   // the same network as SCL:
   "气压故障" := "平衡缸气压检测";
END_REGION

REGION Network 4
   RUNG wire#powerrail
      Contact( "急停故障" )
      Contact( "液压保护故障" )
      Contact( "气压故障" )
      Contact( "润滑正常" )
      Coil( "设备故障" )
   END_RUNG
   // the same network as SCL:
   "设备故障" := "急停故障" AND "液压保护故障" AND "气压故障" AND "润滑正常";
END_REGION
END_FUNCTION

FUNCTION "气垫调整2" : Void   // FC5, LAD
{ S7_Optimized_Access := 'TRUE' }
VERSION : 0.1
BEGIN

REGION Network 2
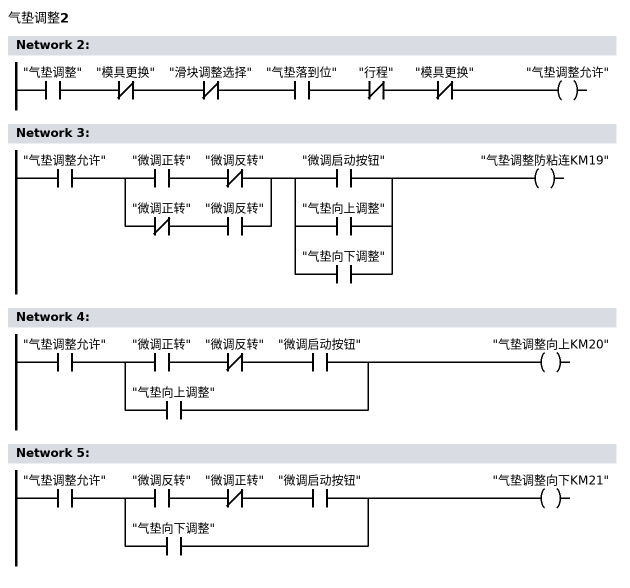
   RUNG wire#powerrail
      Contact( "气垫调整" )
      I_Contact( "模具更换" )
      I_Contact( "滑块调整选择" )
      Contact( "气垫落到位" )
      I_Contact( "行程" )
      I_Contact( "模具更换" )
      Coil( "气垫调整允许" )
   END_RUNG
   // the same network as SCL:
   "气垫调整允许" := "气垫调整" AND NOT "模具更换" AND NOT "滑块调整选择" AND "气垫落到位" AND NOT "行程" AND NOT "模具更换";
END_REGION

REGION Network 3
   RUNG wire#powerrail
      Contact( "气垫调整允许" )
      wire#w1
      Contact( "微调正转" )
      I_Contact( "微调反转" )
      wire#w2
      Contact( "微调启动按钮" )
      wire#w3
      Coil( "气垫调整防粘连KM19" )
   END_RUNG
   RUNG wire#w1
      I_Contact( "微调正转" )
      Contact( "微调反转" )
   END_RUNG wire#w2
   RUNG wire#w2
      Contact( "气垫向上调整" )
   END_RUNG wire#w3
   RUNG wire#w2
      Contact( "气垫向下调整" )
   END_RUNG wire#w3
   // the same network as SCL:
   "气垫调整防粘连KM19" := "气垫调整允许" AND (("微调正转" AND NOT "微调反转") OR (NOT "微调正转" AND "微调反转")) AND ("微调启动按钮" OR "气垫向上调整" OR "气垫向下调整");
END_REGION

REGION Network 4
   RUNG wire#powerrail
      Contact( "气垫调整允许" )
      wire#w1
      Contact( "微调正转" )
      I_Contact( "微调反转" )
      Contact( "微调启动按钮" )
      wire#w2
      Coil( "气垫调整向上KM20" )
   END_RUNG
   RUNG wire#w1
      Contact( "气垫向上调整" )
   END_RUNG wire#w2
   // the same network as SCL:
   "气垫调整向上KM20" := "气垫调整允许" AND (("微调正转" AND NOT "微调反转" AND "微调启动按钮") OR "气垫向上调整");
END_REGION

REGION Network 5
   RUNG wire#powerrail
      Contact( "气垫调整允许" )
      wire#w1
      Contact( "微调反转" )
      I_Contact( "微调正转" )
      Contact( "微调启动按钮" )
      wire#w2
      Coil( "气垫调整向下KM21" )
   END_RUNG
   RUNG wire#w1
      Contact( "气垫向下调整" )
   END_RUNG wire#w2
   // the same network as SCL:
   "气垫调整向下KM21" := "气垫调整允许" AND (("微调反转" AND NOT "微调正转" AND "微调启动按钮") OR "气垫向下调整");
END_REGION
END_FUNCTION

FUNCTION "润滑启动" : Void   // FC6, LAD
{ S7_Optimized_Access := 'TRUE' }
VERSION : 0.1
BEGIN

REGION Network 1
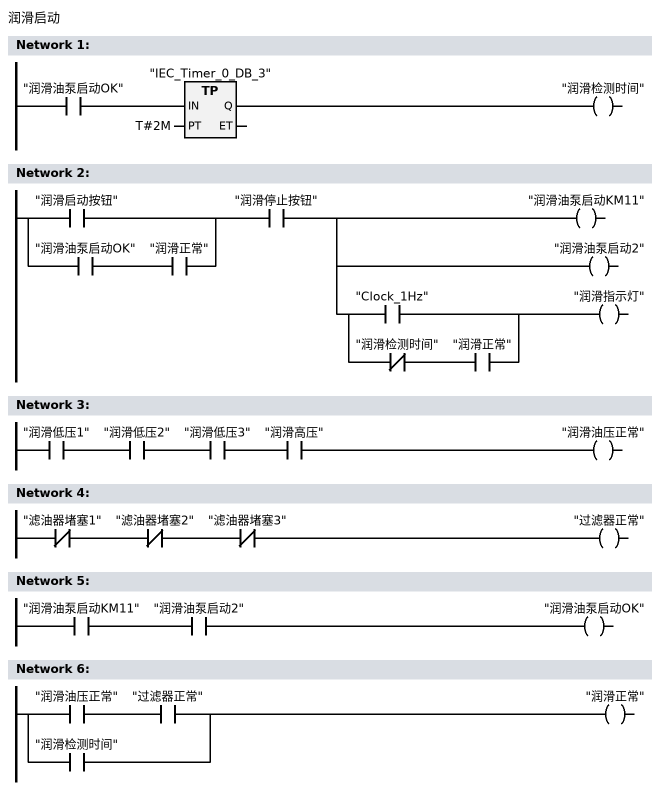
   "IEC_Timer_0_DB_3".TP(IN := "润滑油泵启动OK", PT := T#2M);
   "润滑检测时间" := "IEC_Timer_0_DB_3".Q;
END_REGION

REGION Network 2
   RUNG wire#powerrail
      Contact( "润滑启动按钮" )
      wire#w1
      Contact( "润滑停止按钮" )
      wire#w2
      Coil( "润滑油泵启动KM11" )
   END_RUNG
   RUNG wire#powerrail
      Contact( "润滑油泵启动OK" )
      Contact( "润滑正常" )
   END_RUNG wire#w1
   RUNG wire#w2
      Coil( "润滑油泵启动2" )
   END_RUNG
   RUNG wire#w2
      Contact( "Clock_1Hz" )
      wire#w3
      Coil( "润滑指示灯" )
   END_RUNG
   RUNG wire#w2
      I_Contact( "润滑检测时间" )
      Contact( "润滑正常" )
   END_RUNG wire#w3
   // the same network as SCL:
   "润滑油泵启动KM11" := ("润滑启动按钮" OR ("润滑油泵启动OK" AND "润滑正常")) AND "润滑停止按钮";
   "润滑油泵启动2" := "润滑油泵启动KM11";
   "润滑指示灯" := "润滑油泵启动KM11" AND ("Clock_1Hz" OR (NOT "润滑检测时间" AND "润滑正常"));
END_REGION

REGION Network 3
   RUNG wire#powerrail
      Contact( "润滑低压1" )
      Contact( "润滑低压2" )
      Contact( "润滑低压3" )
      Contact( "润滑高压" )
      Coil( "润滑油压正常" )
   END_RUNG
   // the same network as SCL:
   "润滑油压正常" := "润滑低压1" AND "润滑低压2" AND "润滑低压3" AND "润滑高压";
END_REGION

REGION Network 4
   RUNG wire#powerrail
      I_Contact( "滤油器堵塞1" )
      I_Contact( "滤油器堵塞2" )
      I_Contact( "滤油器堵塞3" )
      Coil( "过滤器正常" )
   END_RUNG
   // the same network as SCL:
   "过滤器正常" := NOT "滤油器堵塞1" AND NOT "滤油器堵塞2" AND NOT "滤油器堵塞3";
END_REGION

REGION Network 5
   RUNG wire#powerrail
      Contact( "润滑油泵启动KM11" )
      Contact( "润滑油泵启动2" )
      Coil( "润滑油泵启动OK" )
   END_RUNG
   // the same network as SCL:
   "润滑油泵启动OK" := "润滑油泵启动KM11" AND "润滑油泵启动2";
END_REGION

REGION Network 6
   RUNG wire#powerrail
      Contact( "润滑油压正常" )
      Contact( "过滤器正常" )
      wire#w1
      Coil( "润滑正常" )
   END_RUNG
   RUNG wire#powerrail
      Contact( "润滑检测时间" )
   END_RUNG wire#w1
   // the same network as SCL:
   "润滑正常" := ("润滑油压正常" AND "过滤器正常") OR "润滑检测时间";
END_REGION
END_FUNCTION

FUNCTION "主电机启动" : Void   // FC7, LAD
{ S7_Optimized_Access := 'TRUE' }
VERSION : 0.1
   VAR_TEMP   // added for the SCL form of the ladder/FBD networks
      _w1 : Bool;
   END_VAR
BEGIN

REGION Network 1
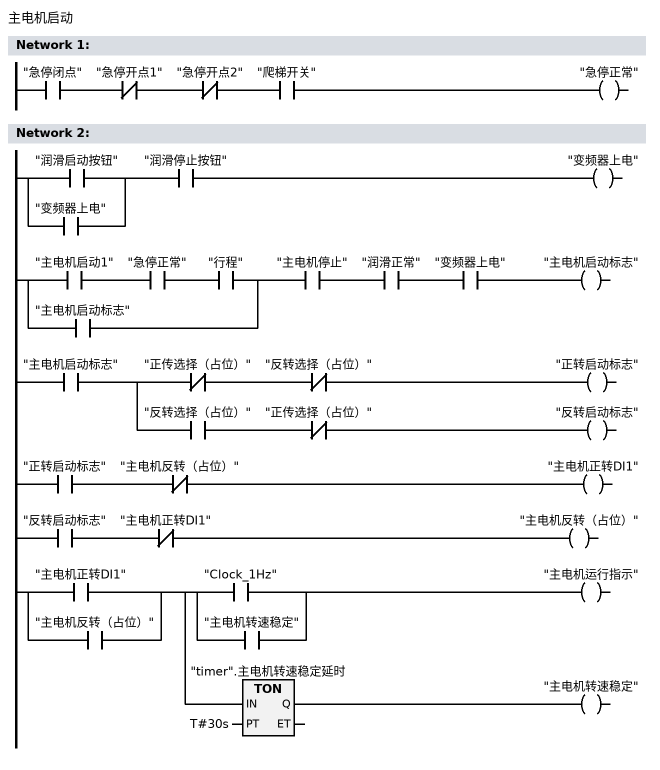
   RUNG wire#powerrail
      Contact( "急停闭点" )
      I_Contact( "急停开点1" )
      I_Contact( "急停开点2" )
      Contact( "爬梯开关" )
      Coil( "急停正常" )
   END_RUNG
   // the same network as SCL:
   "急停正常" := "急停闭点" AND NOT "急停开点1" AND NOT "急停开点2" AND "爬梯开关";
END_REGION

REGION Network 2
   "变频器上电" := ("润滑启动按钮" OR "变频器上电") AND "润滑停止按钮";
   "主电机启动标志" := (("主电机启动1" AND "急停正常" AND "行程") OR "主电机启动标志") AND "主电机停止" AND "润滑正常" AND "变频器上电";
   "正转启动标志" := "主电机启动标志" AND NOT "正传选择（占位）" AND NOT "反转选择（占位）";
   "反转启动标志" := "主电机启动标志" AND "反转选择（占位）" AND NOT "正传选择（占位）";
   "主电机正转DI1" := "正转启动标志" AND NOT "主电机反转（占位）";
   "主电机反转（占位）" := "反转启动标志" AND NOT "主电机正转DI1";
   #_w1 := "主电机正转DI1" OR "主电机反转（占位）";
   "主电机运行指示" := #_w1 AND ("Clock_1Hz" OR "主电机转速稳定");
   "timer".主电机转速稳定延时.TON(IN := #_w1, PT := T#30s);
   "主电机转速稳定" := "timer".主电机转速稳定延时.Q;
END_REGION
END_FUNCTION

FUNCTION "滑块行程" : Void   // FC8, LAD
{ S7_Optimized_Access := 'TRUE' }
VERSION : 0.1
BEGIN

REGION Network 1
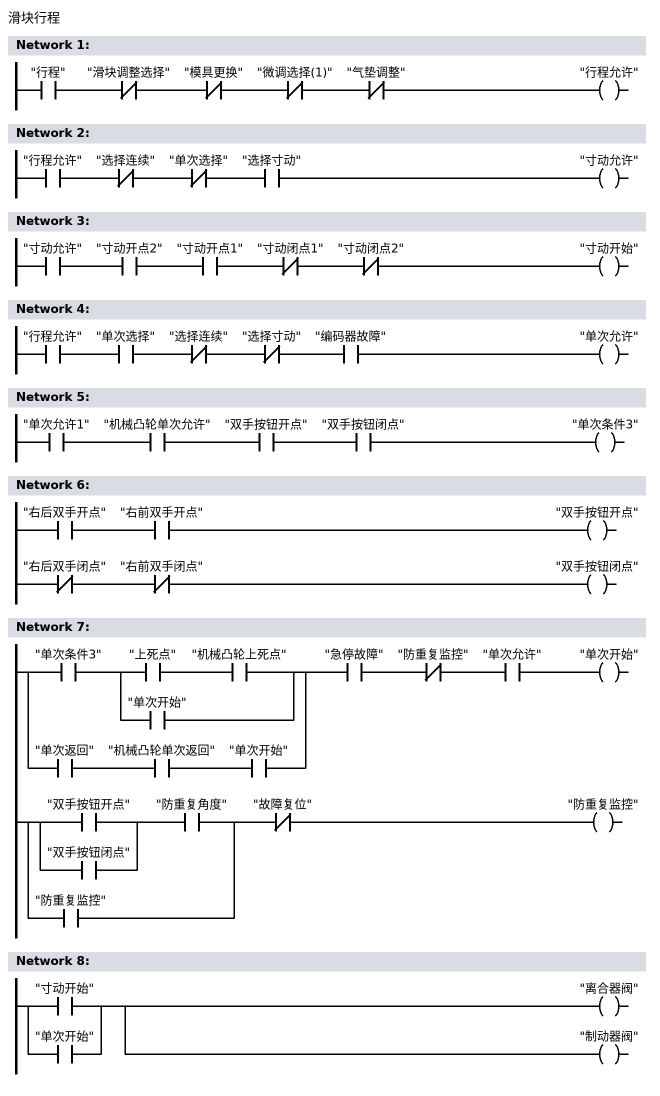
   RUNG wire#powerrail
      Contact( "行程" )
      I_Contact( "滑块调整选择" )
      I_Contact( "模具更换" )
      I_Contact( "微调选择(1)" )
      I_Contact( "气垫调整" )
      Coil( "行程允许" )
   END_RUNG
   // the same network as SCL:
   "行程允许" := "行程" AND NOT "滑块调整选择" AND NOT "模具更换" AND NOT "微调选择(1)" AND NOT "气垫调整";
END_REGION

REGION Network 2
   RUNG wire#powerrail
      Contact( "行程允许" )
      I_Contact( "选择连续" )
      I_Contact( "单次选择" )
      Contact( "选择寸动" )
      Coil( "寸动允许" )
   END_RUNG
   // the same network as SCL:
   "寸动允许" := "行程允许" AND NOT "选择连续" AND NOT "单次选择" AND "选择寸动";
END_REGION

REGION Network 3
   RUNG wire#powerrail
      Contact( "寸动允许" )
      Contact( "寸动开点2" )
      Contact( "寸动开点1" )
      I_Contact( "寸动闭点1" )
      I_Contact( "寸动闭点2" )
      Coil( "寸动开始" )
   END_RUNG
   // the same network as SCL:
   "寸动开始" := "寸动允许" AND "寸动开点2" AND "寸动开点1" AND NOT "寸动闭点1" AND NOT "寸动闭点2";
END_REGION

REGION Network 4
   RUNG wire#powerrail
      Contact( "行程允许" )
      Contact( "单次选择" )
      I_Contact( "选择连续" )
      I_Contact( "选择寸动" )
      Contact( "编码器故障" )
      Coil( "单次允许" )
   END_RUNG
   // the same network as SCL:
   "单次允许" := "行程允许" AND "单次选择" AND NOT "选择连续" AND NOT "选择寸动" AND "编码器故障";
END_REGION

REGION Network 5
   RUNG wire#powerrail
      Contact( "单次允许1" )
      Contact( "机械凸轮单次允许" )
      Contact( "双手按钮开点" )
      Contact( "双手按钮闭点" )
      Coil( "单次条件3" )
   END_RUNG
   // the same network as SCL:
   "单次条件3" := "单次允许1" AND "机械凸轮单次允许" AND "双手按钮开点" AND "双手按钮闭点";
END_REGION

REGION Network 6
   RUNG wire#powerrail
      Contact( "右后双手开点" )
      Contact( "右前双手开点" )
      Coil( "双手按钮开点" )
   END_RUNG
   RUNG wire#powerrail
      I_Contact( "右后双手闭点" )
      I_Contact( "右前双手闭点" )
      Coil( "双手按钮闭点" )
   END_RUNG
   // the same network as SCL:
   "双手按钮开点" := "右后双手开点" AND "右前双手开点";
   "双手按钮闭点" := NOT "右后双手闭点" AND NOT "右前双手闭点";
END_REGION

REGION Network 7
   RUNG wire#powerrail
      Contact( "单次条件3" )
      wire#w1
      Contact( "上死点" )
      Contact( "机械凸轮上死点" )
      wire#w2
      Contact( "急停故障" )
      I_Contact( "防重复监控" )
      Contact( "单次允许" )
      Coil( "单次开始" )
   END_RUNG
   RUNG wire#w1
      Contact( "单次开始" )
   END_RUNG wire#w2
   RUNG wire#powerrail
      Contact( "单次返回" )
      Contact( "机械凸轮单次返回" )
      Contact( "单次开始" )
   END_RUNG wire#w2
   RUNG wire#powerrail
      Contact( "双手按钮开点" )
      wire#w3
      Contact( "防重复角度" )
      wire#w4
      I_Contact( "故障复位" )
      Coil( "防重复监控" )
   END_RUNG
   RUNG wire#powerrail
      Contact( "双手按钮闭点" )
   END_RUNG wire#w3
   RUNG wire#powerrail
      Contact( "防重复监控" )
   END_RUNG wire#w4
   // the same network as SCL:
   "单次开始" := (("单次条件3" AND (("上死点" AND "机械凸轮上死点") OR "单次开始")) OR ("单次返回" AND "机械凸轮单次返回" AND "单次开始")) AND "急停故障" AND NOT "防重复监控" AND "单次允许";
   "防重复监控" := ((("双手按钮开点" OR "双手按钮闭点") AND "防重复角度") OR "防重复监控") AND NOT "故障复位";
END_REGION

REGION Network 8
   RUNG wire#powerrail
      Contact( "寸动开始" )
      wire#w1
      Coil( "离合器阀" )
   END_RUNG
   RUNG wire#powerrail
      Contact( "单次开始" )
   END_RUNG wire#w1
   RUNG wire#w1
      Coil( "制动器阀" )
   END_RUNG
   // the same network as SCL:
   "离合器阀" := "寸动开始" OR "单次开始";
   "制动器阀" := "离合器阀";
END_REGION
END_FUNCTION

FUNCTION "滑块编码器调制" : Void   // FC9, LAD
{ S7_Optimized_Access := 'TRUE' }
VERSION : 0.1
// 滑块编码器
   VAR_TEMP
      D102 : Real;
      D103 : Real;
   END_VAR
BEGIN

REGION Network 1
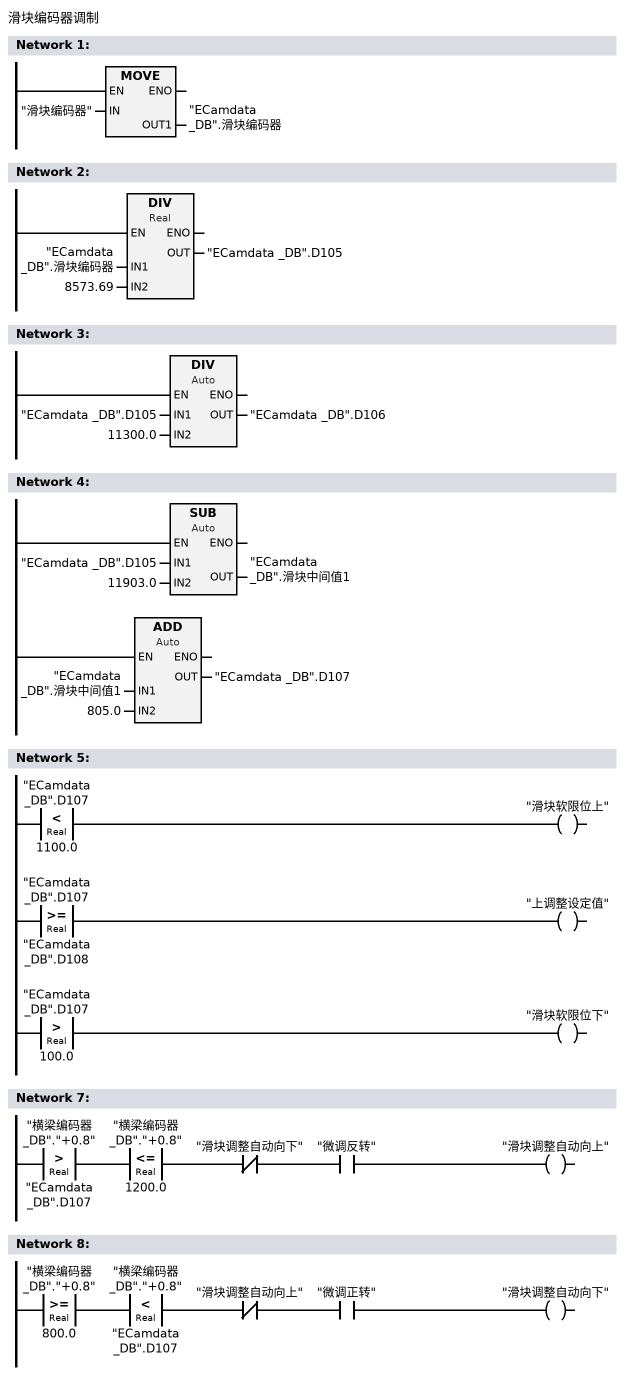
   RUNG wire#powerrail
      Move(in := "滑块编码器", out1 => "ECamdata _DB".滑块编码器)
   END_RUNG
   // the same network as SCL:
   "ECamdata _DB".滑块编码器 := "滑块编码器";
END_REGION

REGION Network 2
   RUNG wire#powerrail
      { S7_Templates := "SrcType := Real" } Div(in1 := "ECamdata _DB".滑块编码器, in2 := 8573.69, out => "ECamdata _DB".D105)
   END_RUNG
   // the same network as SCL:
   "ECamdata _DB".D105 := "ECamdata _DB".滑块编码器 / 8573.69;
END_REGION

REGION Network 3
   RUNG wire#powerrail
      Div(in1 := "ECamdata _DB".D105, in2 := 11300.0, out => "ECamdata _DB".D106)
   END_RUNG
   // the same network as SCL:
   "ECamdata _DB".D106 := "ECamdata _DB".D105 / 11300.0;
END_REGION

REGION Network 4
   RUNG wire#powerrail
      Sub(in1 := "ECamdata _DB".D105, in2 := 11903.0, out => "ECamdata _DB".滑块中间值1)
   END_RUNG
   RUNG wire#powerrail
      Add(in1 := "ECamdata _DB".滑块中间值1, in2 := 805.0, out => "ECamdata _DB".D107)
   END_RUNG
   // the same network as SCL:
   "ECamdata _DB".滑块中间值1 := "ECamdata _DB".D105 - 11903.0;
   "ECamdata _DB".D107 := "ECamdata _DB".滑块中间值1 + 805.0;
END_REGION

REGION Network 5
   RUNG wire#powerrail
      { S7_Templates := "SrcType := Real" } LT_Contact(in1 := "ECamdata _DB".D107, in2 := 1100.0)
      Coil( "滑块软限位上" )
   END_RUNG
   RUNG wire#powerrail
      { S7_Templates := "SrcType := Real" } GE_Contact(in1 := "ECamdata _DB".D107, in2 := "ECamdata _DB".D108)
      Coil( "上调整设定值" )
   END_RUNG
   RUNG wire#powerrail
      { S7_Templates := "SrcType := Real" } GT_Contact(in1 := "ECamdata _DB".D107, in2 := 100.0)
      Coil( "滑块软限位下" )
   END_RUNG
   // the same network as SCL:
   "滑块软限位上" := "ECamdata _DB".D107 < 1100.0;
   "上调整设定值" := "ECamdata _DB".D107 >= "ECamdata _DB".D108;
   "滑块软限位下" := "ECamdata _DB".D107 > 100.0;
END_REGION

REGION Network 7
   RUNG wire#powerrail
      { S7_Templates := "SrcType := Real" } GT_Contact(in1 := "横梁编码器 _DB"."+0.8", in2 := "ECamdata _DB".D107)
      { S7_Templates := "SrcType := Real" } LE_Contact(in1 := "横梁编码器 _DB"."+0.8", in2 := 1200.0)
      I_Contact( "滑块调整自动向下" )
      Contact( "微调反转" )
      Coil( "滑块调整自动向上" )
   END_RUNG
   // the same network as SCL:
   "滑块调整自动向上" := ("横梁编码器 _DB"."+0.8" > "ECamdata _DB".D107) AND ("横梁编码器 _DB"."+0.8" <= 1200.0) AND NOT "滑块调整自动向下" AND "微调反转";
END_REGION

REGION Network 8
   RUNG wire#powerrail
      { S7_Templates := "SrcType := Real" } GE_Contact(in1 := "横梁编码器 _DB"."+0.8", in2 := 800.0)
      { S7_Templates := "SrcType := Real" } LT_Contact(in1 := "横梁编码器 _DB"."+0.8", in2 := "ECamdata _DB".D107)
      I_Contact( "滑块调整自动向上" )
      Contact( "微调正转" )
      Coil( "滑块调整自动向下" )
   END_RUNG
   // the same network as SCL:
   "滑块调整自动向下" := ("横梁编码器 _DB"."+0.8" >= 800.0) AND ("横梁编码器 _DB"."+0.8" < "ECamdata _DB".D107) AND NOT "滑块调整自动向上" AND "微调正转";
END_REGION
END_FUNCTION

FUNCTION "安全报警" : Void   // FC10, LAD
{ S7_Optimized_Access := 'TRUE' }
VERSION : 0.1
BEGIN

REGION Network 1
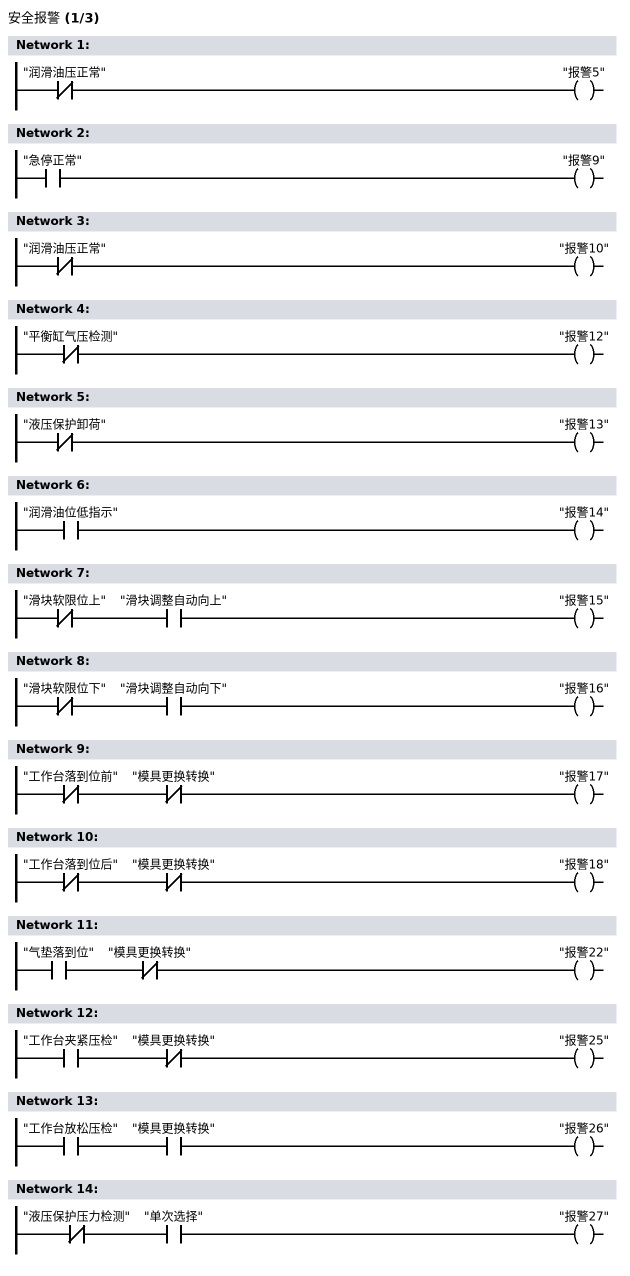
   RUNG wire#powerrail
      I_Contact( "润滑油压正常" )
      Coil( "报警5" )
   END_RUNG
   // the same network as SCL:
   "报警5" := NOT "润滑油压正常";
END_REGION

REGION Network 2
   RUNG wire#powerrail
      Contact( "急停正常" )
      Coil( "报警9" )
   END_RUNG
   // the same network as SCL:
   "报警9" := "急停正常";
END_REGION

REGION Network 3
   RUNG wire#powerrail
      I_Contact( "润滑油压正常" )
      Coil( "报警10" )
   END_RUNG
   // the same network as SCL:
   "报警10" := NOT "润滑油压正常";
END_REGION

REGION Network 4
   RUNG wire#powerrail
      I_Contact( "平衡缸气压检测" )
      Coil( "报警12" )
   END_RUNG
   // the same network as SCL:
   "报警12" := NOT "平衡缸气压检测";
END_REGION

REGION Network 5
   RUNG wire#powerrail
      I_Contact( "液压保护卸荷" )
      Coil( "报警13" )
   END_RUNG
   // the same network as SCL:
   "报警13" := NOT "液压保护卸荷";
END_REGION

REGION Network 6
   RUNG wire#powerrail
      Contact( "润滑油位低指示" )
      Coil( "报警14" )
   END_RUNG
   // the same network as SCL:
   "报警14" := "润滑油位低指示";
END_REGION

REGION Network 7
   RUNG wire#powerrail
      I_Contact( "滑块软限位上" )
      Contact( "滑块调整自动向上" )
      Coil( "报警15" )
   END_RUNG
   // the same network as SCL:
   "报警15" := NOT "滑块软限位上" AND "滑块调整自动向上";
END_REGION

REGION Network 8
   RUNG wire#powerrail
      I_Contact( "滑块软限位下" )
      Contact( "滑块调整自动向下" )
      Coil( "报警16" )
   END_RUNG
   // the same network as SCL:
   "报警16" := NOT "滑块软限位下" AND "滑块调整自动向下";
END_REGION

REGION Network 9
   RUNG wire#powerrail
      I_Contact( "工作台落到位前" )
      I_Contact( "模具更换转换" )
      Coil( "报警17" )
   END_RUNG
   // the same network as SCL:
   "报警17" := NOT "工作台落到位前" AND NOT "模具更换转换";
END_REGION

REGION Network 10
   RUNG wire#powerrail
      I_Contact( "工作台落到位后" )
      I_Contact( "模具更换转换" )
      Coil( "报警18" )
   END_RUNG
   // the same network as SCL:
   "报警18" := NOT "工作台落到位后" AND NOT "模具更换转换";
END_REGION

REGION Network 11
   RUNG wire#powerrail
      Contact( "气垫落到位" )
      I_Contact( "模具更换转换" )
      Coil( "报警22" )
   END_RUNG
   // the same network as SCL:
   "报警22" := "气垫落到位" AND NOT "模具更换转换";
END_REGION

REGION Network 12
   RUNG wire#powerrail
      Contact( "工作台夹紧压检" )
      I_Contact( "模具更换转换" )
      Coil( "报警25" )
   END_RUNG
   // the same network as SCL:
   "报警25" := "工作台夹紧压检" AND NOT "模具更换转换";
END_REGION

REGION Network 13
   RUNG wire#powerrail
      Contact( "工作台放松压检" )
      Contact( "模具更换转换" )
      Coil( "报警26" )
   END_RUNG
   // the same network as SCL:
   "报警26" := "工作台放松压检" AND "模具更换转换";
END_REGION

REGION Network 14
   RUNG wire#powerrail
      I_Contact( "液压保护压力检测" )
      Contact( "单次选择" )
      Coil( "报警27" )
   END_RUNG
   // the same network as SCL:
   "报警27" := NOT "液压保护压力检测" AND "单次选择";
END_REGION

REGION Network 15
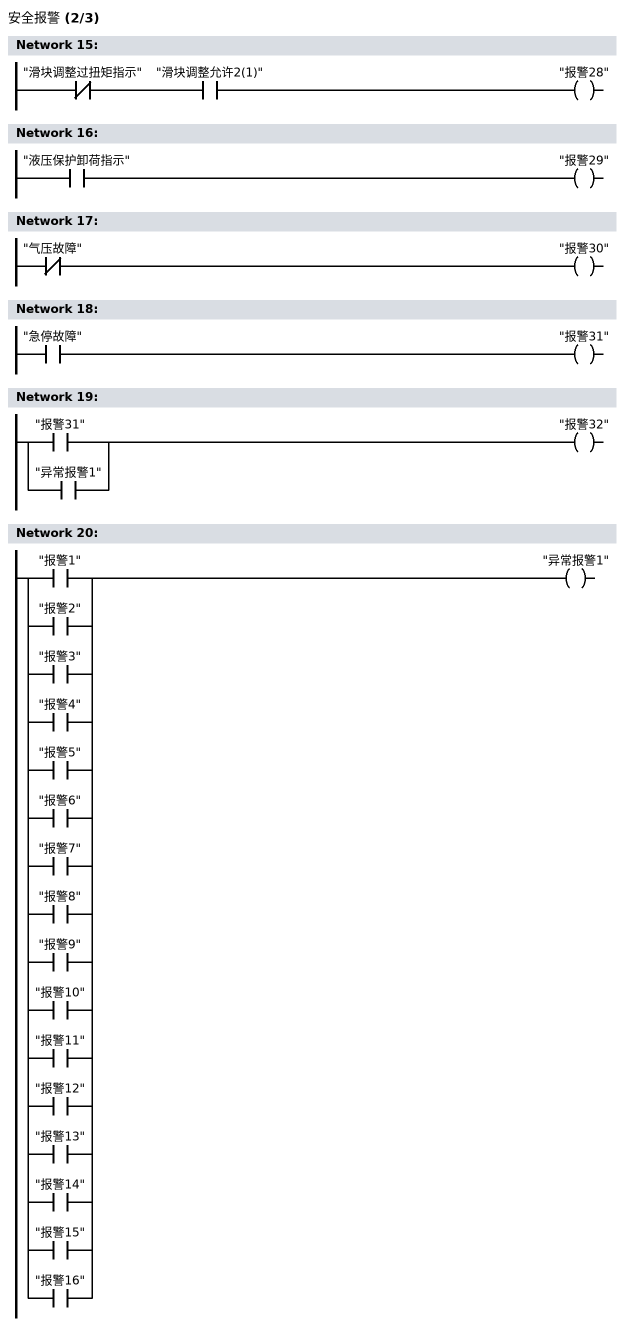
   RUNG wire#powerrail
      I_Contact( "滑块调整过扭矩指示" )
      Contact( "滑块调整允许2(1)" )
      Coil( "报警28" )
   END_RUNG
   // the same network as SCL:
   "报警28" := NOT "滑块调整过扭矩指示" AND "滑块调整允许2(1)";
END_REGION

REGION Network 16
   RUNG wire#powerrail
      Contact( "液压保护卸荷指示" )
      Coil( "报警29" )
   END_RUNG
   // the same network as SCL:
   "报警29" := "液压保护卸荷指示";
END_REGION

REGION Network 17
   RUNG wire#powerrail
      I_Contact( "气压故障" )
      Coil( "报警30" )
   END_RUNG
   // the same network as SCL:
   "报警30" := NOT "气压故障";
END_REGION

REGION Network 18
   RUNG wire#powerrail
      Contact( "急停故障" )
      Coil( "报警31" )
   END_RUNG
   // the same network as SCL:
   "报警31" := "急停故障";
END_REGION

REGION Network 19
   RUNG wire#powerrail
      Contact( "报警31" )
      wire#w1
      Coil( "报警32" )
   END_RUNG
   RUNG wire#powerrail
      Contact( "异常报警1" )
   END_RUNG wire#w1
   // the same network as SCL:
   "报警32" := "报警31" OR "异常报警1";
END_REGION

REGION Network 20
   RUNG wire#powerrail
      Contact( "报警1" )
      wire#w1
      Coil( "异常报警1" )
   END_RUNG
   RUNG wire#powerrail
      Contact( "报警2" )
   END_RUNG wire#w1
   RUNG wire#powerrail
      Contact( "报警3" )
   END_RUNG wire#w1
   RUNG wire#powerrail
      Contact( "报警4" )
   END_RUNG wire#w1
   RUNG wire#powerrail
      Contact( "报警5" )
   END_RUNG wire#w1
   RUNG wire#powerrail
      Contact( "报警6" )
   END_RUNG wire#w1
   RUNG wire#powerrail
      Contact( "报警7" )
   END_RUNG wire#w1
   RUNG wire#powerrail
      Contact( "报警8" )
   END_RUNG wire#w1
   RUNG wire#powerrail
      Contact( "报警9" )
   END_RUNG wire#w1
   RUNG wire#powerrail
      Contact( "报警10" )
   END_RUNG wire#w1
   RUNG wire#powerrail
      Contact( "报警11" )
   END_RUNG wire#w1
   RUNG wire#powerrail
      Contact( "报警12" )
   END_RUNG wire#w1
   RUNG wire#powerrail
      Contact( "报警13" )
   END_RUNG wire#w1
   RUNG wire#powerrail
      Contact( "报警14" )
   END_RUNG wire#w1
   RUNG wire#powerrail
      Contact( "报警15" )
   END_RUNG wire#w1
   RUNG wire#powerrail
      Contact( "报警16" )
   END_RUNG wire#w1
   // the same network as SCL:
   "异常报警1" := "报警1" OR "报警2" OR "报警3" OR "报警4" OR "报警5" OR "报警6" OR "报警7" OR "报警8" OR "报警9" OR "报警10" OR "报警11" OR "报警12" OR "报警13" OR "报警14" OR "报警15" OR "报警16";
END_REGION

REGION Network 21
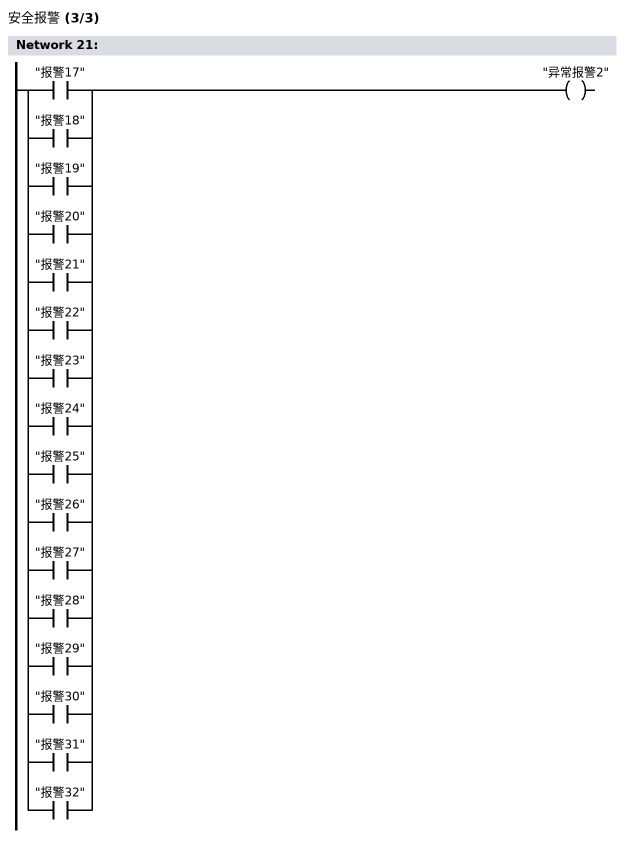
   RUNG wire#powerrail
      Contact( "报警17" )
      wire#w1
      Coil( "异常报警2" )
   END_RUNG
   RUNG wire#powerrail
      Contact( "报警18" )
   END_RUNG wire#w1
   RUNG wire#powerrail
      Contact( "报警19" )
   END_RUNG wire#w1
   RUNG wire#powerrail
      Contact( "报警20" )
   END_RUNG wire#w1
   RUNG wire#powerrail
      Contact( "报警21" )
   END_RUNG wire#w1
   RUNG wire#powerrail
      Contact( "报警22" )
   END_RUNG wire#w1
   RUNG wire#powerrail
      Contact( "报警23" )
   END_RUNG wire#w1
   RUNG wire#powerrail
      Contact( "报警24" )
   END_RUNG wire#w1
   RUNG wire#powerrail
      Contact( "报警25" )
   END_RUNG wire#w1
   RUNG wire#powerrail
      Contact( "报警26" )
   END_RUNG wire#w1
   RUNG wire#powerrail
      Contact( "报警27" )
   END_RUNG wire#w1
   RUNG wire#powerrail
      Contact( "报警28" )
   END_RUNG wire#w1
   RUNG wire#powerrail
      Contact( "报警29" )
   END_RUNG wire#w1
   RUNG wire#powerrail
      Contact( "报警30" )
   END_RUNG wire#w1
   RUNG wire#powerrail
      Contact( "报警31" )
   END_RUNG wire#w1
   RUNG wire#powerrail
      Contact( "报警32" )
   END_RUNG wire#w1
   // the same network as SCL:
   "异常报警2" := "报警17" OR "报警18" OR "报警19" OR "报警20" OR "报警21" OR "报警22" OR "报警23" OR "报警24" OR "报警25" OR "报警26" OR "报警27" OR "报警28" OR "报警29" OR "报警30" OR "报警31" OR "报警32";
END_REGION
END_FUNCTION

FUNCTION "液压保护" : Void   // FC11, LAD
{ S7_Optimized_Access := 'TRUE' }
VERSION : 0.1
BEGIN

REGION Network 1
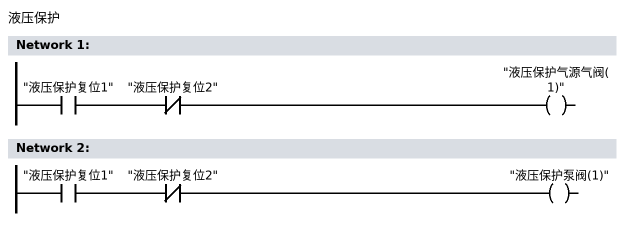
   RUNG wire#powerrail
      Contact( "液压保护复位1" )
      I_Contact( "液压保护复位2" )
      Coil( "液压保护气源气阀(1)" )
   END_RUNG
   // the same network as SCL:
   "液压保护气源气阀(1)" := "液压保护复位1" AND NOT "液压保护复位2";
END_REGION

REGION Network 2
   RUNG wire#powerrail
      Contact( "液压保护复位1" )
      I_Contact( "液压保护复位2" )
      Coil( "液压保护泵阀(1)" )
   END_RUNG
   // the same network as SCL:
   "液压保护泵阀(1)" := "液压保护复位1" AND NOT "液压保护复位2";
END_REGION
END_FUNCTION

FUNCTION "产品计数" : Void   // FC12, LAD
{ S7_Optimized_Access := 'TRUE' }
VERSION : 0.1
   VAR_TEMP
      气垫位置 : DB_ANY;
   END_VAR
BEGIN

REGION Network 1
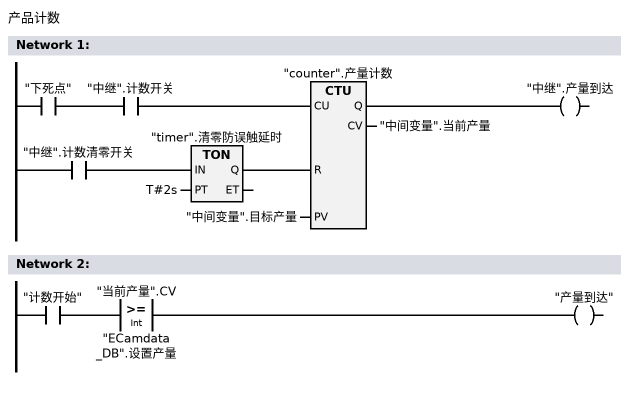
   "timer".清零防误触延时.TON(IN := "中继".计数清零开关, PT := T#2s);
   "counter".产量计数.CTU(CU := "下死点" AND "中继".计数开关, R := "timer".清零防误触延时.Q, PV := "中间变量".目标产量, CV => "中间变量".当前产量);
   "中继".产量到达 := "counter".产量计数.Q;
END_REGION

REGION Network 2
   RUNG wire#powerrail
      Contact( "计数开始" )
      { S7_Templates := "SrcType := Int" } GE_Contact(in1 := "当前产量".CV, in2 := "ECamdata _DB".设置产量)
      Coil( "产量到达" )
   END_RUNG
   // the same network as SCL:
   "产量到达" := "计数开始" AND ("当前产量".CV >= "ECamdata _DB".设置产量);
END_REGION
END_FUNCTION

FUNCTION "通讯诊断" : Void   // FC13, LAD
{ S7_Optimized_Access := 'TRUE' }
VERSION : 0.1
BEGIN

REGION Network 1: 横梁编码器诊断
   // 横梁编码器诊断
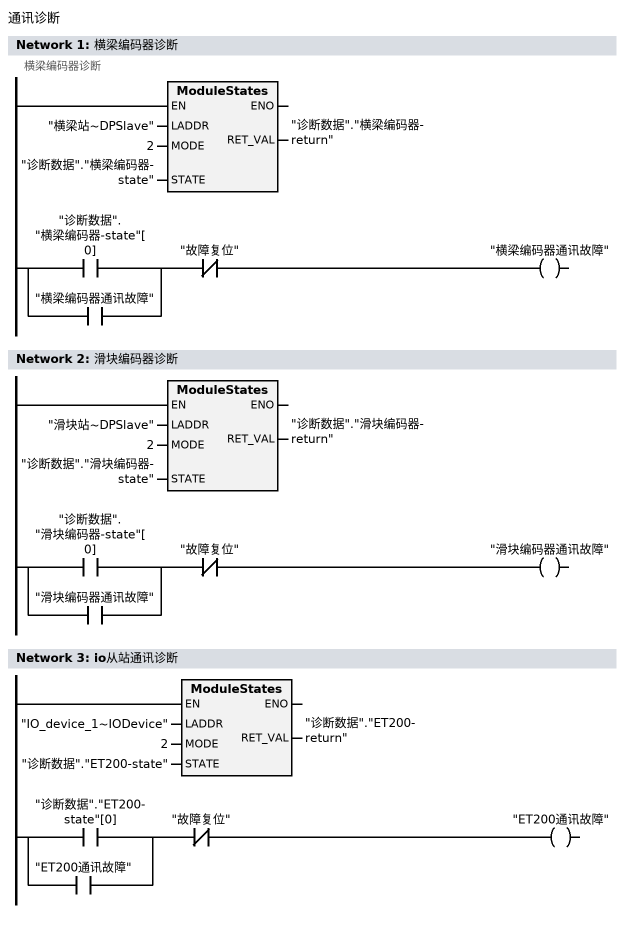
   // no SCL statement known for ModuleStates: written as a call
   "诊断数据"."横梁编码器-return" := ModuleStates(LADDR := "横梁站~DPSlave", MODE := 2, STATE := "诊断数据"."横梁编码器-state");
   "横梁编码器通讯故障" := ("诊断数据"."横梁编码器-state"[0] OR "横梁编码器通讯故障") AND NOT "故障复位";
END_REGION

REGION Network 2: 滑块编码器诊断
   // no SCL statement known for ModuleStates: written as a call
   "诊断数据"."滑块编码器-return" := ModuleStates(LADDR := "滑块站~DPSlave", MODE := 2, STATE := "诊断数据"."滑块编码器-state");
   "滑块编码器通讯故障" := ("诊断数据"."滑块编码器-state"[0] OR "滑块编码器通讯故障") AND NOT "故障复位";
END_REGION

REGION Network 3: io从站通讯诊断
   // no SCL statement known for ModuleStates: written as a call
   "诊断数据"."ET200-return" := ModuleStates(LADDR := "IO_device_1~IODevice",
                           MODE := 2,
                           STATE := "诊断数据"."ET200-state");
   "ET200通讯故障" := ("诊断数据"."ET200-state"[0] OR "ET200通讯故障") AND NOT "故障复位";
END_REGION
END_FUNCTION

ORGANIZATION_BLOCK "IO测试"   // OB125, LAD, ProgramCycle
TITLE = "Main Program Sweep (Cycle)"
{ S7_Optimized_Access := 'TRUE' }
VERSION : 0.1
   VAR_INPUT
      Initial_Call : Bool;   // Initial call of this OB
      Remanence : Bool;   // =True, if remanent data are available
   END_VAR
BEGIN
END_ORGANIZATION_BLOCK

ORGANIZATION_BLOCK "Main"   // OB129, LAD, ProgramCycle
TITLE = "Main Program Sweep (Cycle)"
{ S7_Optimized_Access := 'TRUE' }
VERSION : 0.1
   VAR_INPUT
      Initial_Call : Bool;   // Initial call of this OB
      Remanence : Bool;   // =True, if remanent data are available
   END_VAR
BEGIN

REGION Network 1
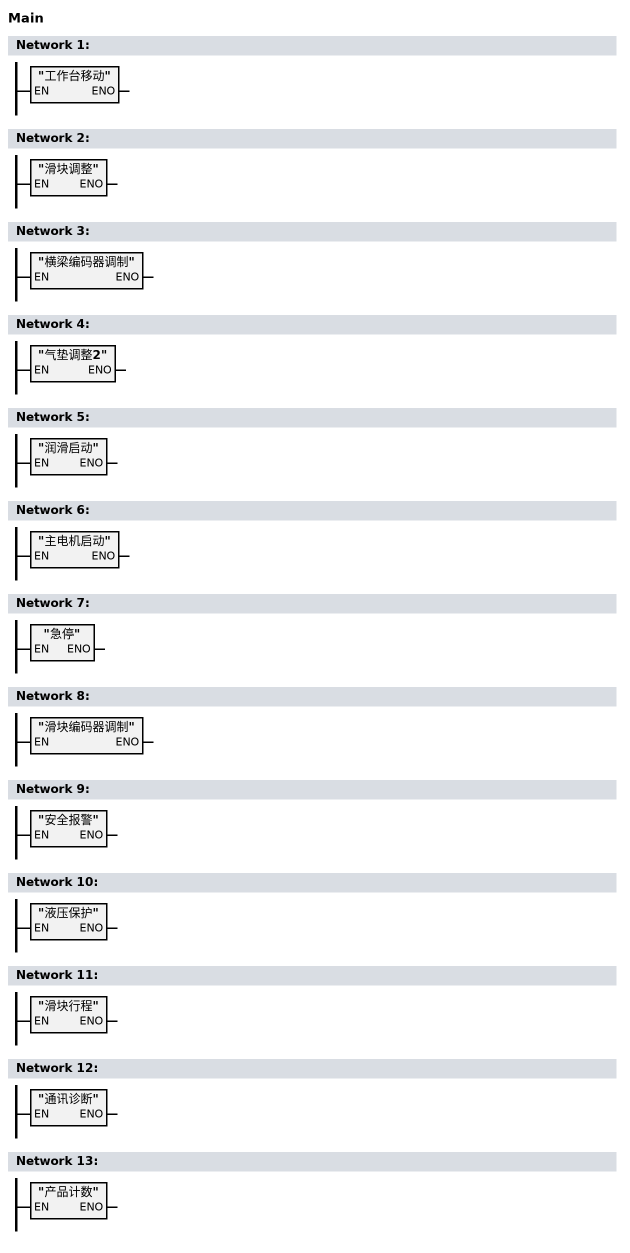
   RUNG wire#powerrail
      "工作台移动"()
   END_RUNG
   // the same network as SCL:
   "工作台移动"();
END_REGION

REGION Network 2
   RUNG wire#powerrail
      "滑块调整"()
   END_RUNG
   // the same network as SCL:
   "滑块调整"();
END_REGION

REGION Network 3
   RUNG wire#powerrail
      "横梁编码器调制"()
   END_RUNG
   // the same network as SCL:
   "横梁编码器调制"();
END_REGION

REGION Network 4
   RUNG wire#powerrail
      "气垫调整2"()
   END_RUNG
   // the same network as SCL:
   "气垫调整2"();
END_REGION

REGION Network 5
   RUNG wire#powerrail
      "润滑启动"()
   END_RUNG
   // the same network as SCL:
   "润滑启动"();
END_REGION

REGION Network 6
   RUNG wire#powerrail
      "主电机启动"()
   END_RUNG
   // the same network as SCL:
   "主电机启动"();
END_REGION

REGION Network 7
   RUNG wire#powerrail
      "急停"()
   END_RUNG
   // the same network as SCL:
   "急停"();
END_REGION

REGION Network 8
   RUNG wire#powerrail
      "滑块编码器调制"()
   END_RUNG
   // the same network as SCL:
   "滑块编码器调制"();
END_REGION

REGION Network 9
   RUNG wire#powerrail
      "安全报警"()
   END_RUNG
   // the same network as SCL:
   "安全报警"();
END_REGION

REGION Network 10
   RUNG wire#powerrail
      "液压保护"()
   END_RUNG
   // the same network as SCL:
   "液压保护"();
END_REGION

REGION Network 11
   RUNG wire#powerrail
      "滑块行程"()
   END_RUNG
   // the same network as SCL:
   "滑块行程"();
END_REGION

REGION Network 12
   RUNG wire#powerrail
      "通讯诊断"()
   END_RUNG
   // the same network as SCL:
   "通讯诊断"();
END_REGION

REGION Network 13
   RUNG wire#powerrail
      "产品计数"()
   END_RUNG
   // the same network as SCL:
   "产品计数"();
END_REGION
END_ORGANIZATION_BLOCK

(* ===== HMI "HMI_RT_1" =====
system functions are stored by id; their names below are inferred from use
connection "HMI_连接_1": ETHERNET, S7_1200_OMS

HMI tags "默认变量表"
   "主电机运行指示" : Bool = PLC 主电机运行指示 AT %Q11.2, 100 ms
   "滑块向上" : Bool = PLC 滑块向上 AT %I14.5, 1 s
   "滑块向下KM7" : Bool = PLC 滑块向下KM7 AT %Q3.2, 1 s
   "滑块向上KM6" : Bool = PLC 滑块向上KM6 AT %Q3.1, 1 s
   "360" : Bool = PLC 360 AT %M204.3, 100 ms
   "10度" : Bool = PLC 10度 AT %M200.0, 100 ms
   "20度" : Bool = PLC 20度 AT %M200.1, 100 ms
   "30度" : Bool = PLC 30度 AT %M200.2, 100 ms
   "40度" : Bool = PLC 40度 AT %M200.3, 100 ms
   "50" : Bool = PLC 50 AT %M200.4, 100 ms
   "60" : Bool = PLC 60 AT %M200.5, 100 ms
   "70" : Bool = PLC 70 AT %M200.6, 100 ms
   "80" : Bool = PLC 80 AT %M200.7, 100 ms
   "90" : Bool = PLC 90 AT %M201.0, 100 ms
   "100" : Bool = PLC 100 AT %M201.1, 100 ms
   "110" : Bool = PLC 110 AT %M201.2, 100 ms
   "120" : Bool = PLC 120 AT %M201.3, 100 ms
   "130" : Bool = PLC 130 AT %M201.4, 100 ms
   "140" : Bool, internal
   "150" : Bool = PLC 150 AT %M201.6, 100 ms
   "160" : Bool = PLC 160 AT %M201.7, 100 ms
   "170" : Bool = PLC 170 AT %M202.0, 100 ms
   "180" : Bool = PLC 180 AT %M202.1, 100 ms
   "190" : Bool = PLC 190 AT %M202.2, 100 ms
   "200" : Bool = PLC 200 AT %M202.3, 100 ms
   "210" : Bool = PLC 210 AT %M202.4, 100 ms
   "220" : Bool = PLC 220 AT %M202.5, 100 ms
   "230" : Bool = PLC 230 AT %M202.6, 100 ms
   "240" : Bool = PLC 240 AT %M202.7, 100 ms
   "250" : Bool = PLC 250 AT %M203.0, 100 ms
   "260" : Bool = PLC 260 AT %M203.1, 100 ms
   "270" : Bool = PLC 270 AT %M203.2, 100 ms
   "280" : Bool = PLC 280 AT %M203.3, 100 ms
   "290" : Bool = PLC 290 AT %M203.4, 100 ms
   "300" : Bool = PLC 300 AT %M203.5, 100 ms
   "310" : Bool = PLC 310 AT %M203.6, 100 ms
   "320" : Bool = PLC 320 AT %M203.7, 100 ms
   "330" : Bool = PLC 330 AT %M204.0, 100 ms
   "340" : Bool = PLC 340 AT %M204.1, 100 ms
   "350" : Bool = PLC 350 AT %M204.2, 100 ms
   "工作台落到位前" : Bool = PLC "Tag_57(1)" AT %I7.3, 1 s
   "工作台落到位后" : Bool = PLC "Tag_58(1)" AT %I7.4, 1 s
   "工作台夹紧压检" : Bool = PLC 工作台夹紧压检 AT %I18.0, 1 s
   "工作台夹紧阀(1)" : Bool = PLC "工作台夹紧阀(1)" AT %Q13.1, 1 s
   "平衡缸气压检测" : Bool = PLC 平衡缸气压检测 AT %I15.6, 1 s
   "润滑油泵启动OK" : Bool = PLC 润滑油泵启动OK AT %M5.5, 1 s
   "润滑油压正常" : Bool = PLC 润滑油压正常 AT %M5.1, 1 s
   "滤油器堵塞指示" : Bool = PLC 滤油器堵塞指示 AT %Q10.5, 1 s
   "急停开点左后" : Bool = PLC "Tag_45(1)" AT %I5.7, 1 s
   "急停开点左前" : Bool = PLC "Tag_44(1)" AT %I5.6, 1 s
   "爬梯开关" : Bool = PLC 爬梯开关 AT %I15.5, 1 s
   "液压保护压力检测" : Bool = PLC 液压保护压力检测 AT %I15.3, 1 s
   "液压保护卸荷" : Bool = PLC 液压保护卸荷 AT %I15.2, 1 s
   "液压保护故障" : Bool = PLC 液压保护故障 AT %M6.1, 1 s
   "横梁编码器" : DWord = PLC 横梁编码器 AT %ID68, 1 s
   "ECamdata _DB_+0.7" : DInt = PLC 滑块编码器 AT %ID72, 1 s
   "横梁编码器 _DB_+0.6" : Int = PLC "横梁编码器 _DB"."角度校准值(原+0.6）", 1 s
   "上死点指示" : Bool = PLC 上死点指示 AT %Q10.1, 1 s
   "工作台松开" : Bool = PLC 工作台松开 AT %I11.3, 1 s
   "工作台放松阀(1)" : Bool = PLC "工作台放松阀(1)" AT %Q13.2, 1 s
   "工作台放松压检" : Bool = PLC 工作台放松压检 AT %I18.1, 1 s
   "工作台落到位" : Bool = PLC 工作台落到位 AT %M7.1, 1 s
   "工作台夹紧" : Bool = PLC 工作台夹紧 AT %I11.2, 1 s
   "工作台-夹紧OK" : Bool = PLC "工作台-夹紧OK" AT %M15.2, 1 s
   "工作台放松OK" : Bool = PLC 工作台放松OK AT %M15.3, 1 s
   "横梁编码器 _DB_0.11" : Real = PLC "横梁编码器 _DB"."0.11", 1 s
   "滑块调整自动选择" : Bool = PLC 滑块调整自动选择 AT %M16.2, 1 s
   "ECamdata _DB_+0.36" : Int = PLC "ECamdata _DB"."+0.36", 100 ms
   "ECamdata _DB_+0.47" : Real = PLC "ECamdata _DB"."+0.47", 100 ms
   "ECamdata _DB_+0.6" : Int = PLC "ECamdata _DB".电子凸轮编码器显示, 100 ms
   "ECamdata _DB_AQD" : Real = PLC "ECamdata _DB".平衡器压力显示, 100 ms
   "ECamdata _DB_AQD2" : Real = PLC "ECamdata _DB".AQD2, 100 ms
   "ECamdata _DB_AQD3" : Real = PLC "ECamdata _DB".气垫模拟量显示1, 100 ms
   "ECamdata _DB_D{0}" : Real = PLC "ECamdata _DB".D[0], 100 ms
   "ECamdata _DB_D{1}" : Real = PLC "ECamdata _DB".D[1], 100 ms
   "ECamdata _DB_D{10}滑块设定高度" : Real = PLC "ECamdata _DB".D[10], 100 ms
   "ECamdata _DB_D{11}" : Real = PLC "ECamdata _DB".D[11], 100 ms
   "ECamdata _DB_D{6}" : Real = PLC "ECamdata _DB".D[6], 100 ms
   "ECamdata _DB_D{7}" : Real = PLC "ECamdata _DB".D[7], 100 ms
   "ECamdata _DB_D{9}" : Real = PLC "ECamdata _DB".D[9], 100 ms
   "ECamdata _DB_D102" : Int = PLC "ECamdata _DB".D102, 100 ms
   "ECamdata _DB_D107" : Int = PLC "ECamdata _DB".D107, 100 ms
   "ECamdata _DB_D108" : Real = PLC "ECamdata _DB".D108, 1 s
   "ECamdata _DB_当前产量" : Int = PLC "ECamdata _DB".当前产量, 1 s
   "ECamdata _DB_滑块打油次数" : Int = PLC "ECamdata _DB".滑块打油次数, 100 ms
   "ECamdata _DB_平衡器设置压力" : Real = PLC "ECamdata _DB".平衡器设置压力, 100 ms
   "ECamdata _DB_气垫2压力设置" : Real = PLC "ECamdata _DB".气垫2压力设置, 100 ms
   "ECamdata _DB_气垫模拟量显示1" : Real = PLC "ECamdata _DB".气垫模拟量显示2, 100 ms
   "ECamdata _DB_气垫压力设置" : Real = PLC "ECamdata _DB".气垫1压力设置, 100 ms
   "ECamdata _DB_设置产量" : Int = PLC "ECamdata _DB".设置产量, 1 s
   "ECamdata _DB_主分油器打油次数" : Int = PLC "ECamdata _DB".主分油器打油次数, 100 ms
   "滑块调整手动/自动" : Bool = PLC "滑块调整手动/自动" AT %M301.5, 100 ms
   "ECamdata _DB_D{10}滑块设定高度(1)" : Real = PLC "ECamdata _DB_D{10}滑块设定高度" AT %MD150, 1 s
   "横梁编码器 _DB_+0.8" : Int = PLC "横梁编码器 _DB"."+0.8", 1 s
   "PLC报警变量组1" : Int = PLC PLC报警变量组1 AT %MW3000, 1 s
   "PLC报警变量组2" : Int = PLC PLC报警变量组2 AT %MW3002, 1 s
   "气垫落到位" : Bool = PLC 气垫落到位 AT %I17.5, 1 s
   "工作台落到位后(1)" : Bool = PLC 工作台落到位后 AT %I17.4, 1 s
   "气垫调整" : Bool = PLC 气垫调整 AT %I14.3, 1 s
   "气垫调整向上KM20" : Bool = PLC 气垫调整向上KM20 AT %Q2.5, 1 s
   "气垫调整向下KM21" : Bool = PLC 气垫调整向下KM21 AT %Q2.6, 1 s
   "气垫向上调整" : Bool = PLC 气垫向上调整 AT %M220.0, 1 s
   "气垫向下调整" : Bool = PLC 气垫向下调整 AT %M220.1, 1 s
   "计数清零" : Bool = PLC 计数清零 AT %M30.1, 1 s
   "计数开始" : Bool = PLC 计数开始 AT %M30.0, 1 s
   "当前产量" : Int = PLC 当前产量.CV, 1 s
   "产量到达" : Bool = PLC 产量到达 AT %M30.2, 1 s
   "上死点" : Bool = PLC 上死点 AT %M204.4, 1 s
   "下死点" : Bool = PLC 下死点 AT %M204.6, 1 s
   "故障复位" : Bool = PLC 故障复位 AT %I12.4, 1 s
   "主电机启动接触器接通" : Bool = PLC 主电机启动接触器接通 AT %I3.5, 1 s
   "滑块调整选择" : Bool = PLC 滑块调整选择 AT %I14.1, 1 s
   "行程" : Bool = PLC 行程 AT %I14.2, 1 s
   "模具更换" : Bool = PLC 模具更换 AT %I14.4, 1 s
   "滑块向下" : Bool = PLC 滑块向下 AT %I14.6, 1 s
   "停上死点" : Bool = PLC 停上死点 AT %I14.7, 1 s
   "滑块调整过扭矩" : Bool = PLC 滑块调整过扭矩 AT %I15.1, 1 s
   "润滑停止按钮" : Bool = PLC 润滑停止按钮 AT %I10.0, 1 s
   "润滑启动按钮" : Bool = PLC 润滑启动按钮 AT %I10.1, 1 s
   "气垫手动润滑按钮" : Bool = PLC 气垫手动润滑按钮 AT %I10.2, 1 s
   "平衡缸手动润滑按钮" : Bool = PLC 平衡缸手动润滑按钮 AT %I10.3, 1 s
   "液压保护复位1" : Bool = PLC 液压保护复位1 AT %I10.5, 1 s
   "液压保护复位2" : Bool = PLC 液压保护复位2 AT %I10.6, 1 s
   "模具夹紧按钮" : Bool = PLC 模具夹紧按钮 AT %I10.7, 1 s
   "模具松开按钮" : Bool = PLC 模具松开按钮 AT %I11.0, 1 s
   "模具更换转换" : Bool = PLC 模具更换转换 AT %I11.1, 1 s
   "微调启动按钮" : Bool = PLC 微调启动按钮 AT %I11.4, 1 s
   "微调正转" : Bool = PLC 微调正转 AT %I11.5, 1 s
   "微调反转" : Bool = PLC 微调反转 AT %I11.6, 1 s
   "主电机停止" : Bool = PLC 主电机停止 AT %I11.7, 1 s
   "主电机启动1" : Bool = PLC 主电机启动1 AT %I12.0, 1 s
   "微调选择(1)" : Bool = PLC "微调选择(1)" AT %I14.0, 1 s
   "主电机启动2" : Bool = PLC 主电机启动2 AT %I12.1, 1 s
   "寸动开点1" : Bool = PLC 寸动开点1 AT %I12.2, 1 s
   "寸动闭点1" : Bool = PLC 寸动闭点1 AT %I12.3, 1 s
   "寸动开点2" : Bool = PLC 寸动开点2 AT %I12.5, 1 s
   "寸动闭点2" : Bool = PLC 寸动闭点2 AT %I12.6, 1 s
   "寸动选择" : Bool = PLC 选择连续 AT %I13.1, 1 s
   "单次选择" : Bool = PLC 单次选择 AT %I13.2, 1 s
   "连续选择" : Bool = PLC 选择寸动 AT %I13.3, 1 s
   "急停闭点" : Bool = PLC 急停闭点 AT %I13.5, 1 s
   "急停开点1" : Bool = PLC 急停开点1 AT %I13.6, 1 s
   "急停开点2" : Bool = PLC 急停开点2 AT %I13.7, 1 s
   "润滑油位高" : Bool = PLC 润滑油位高 AT %I16.0, 1 s
   "润滑油位低" : Bool = PLC 润滑油位低 AT %I16.1, 1 s
   "润滑低压1" : Bool = PLC 润滑低压1 AT %I16.3, 1 s
   "润滑低压2" : Bool = PLC 润滑低压2 AT %I16.4, 1 s
   "润滑低压3" : Bool = PLC 润滑低压3 AT %I16.5, 1 s
   "润滑高压" : Bool = PLC 润滑高压 AT %I16.6, 1 s
   "滤油器堵塞1" : Bool = PLC 滤油器堵塞1 AT %I16.7, 1 s
   "滤油器堵塞2" : Bool = PLC 滤油器堵塞2 AT %I17.0, 1 s
   "滤油器堵塞3" : Bool = PLC 滤油器堵塞3 AT %I17.1, 1 s
   "工作台落到位前(1)" : Bool = PLC 工作台落到位前 AT %I17.3, 1 s
   "主电机正转DI1" : Bool = PLC 主电机正转DI1 AT %Q1.0, 1 s
   "润滑油泵启动2" : Bool = PLC 润滑油泵启动2 AT %Q2.0, 1 s
   "M6 ?" : Bool = PLC "M6 ?" AT %Q2.1, 1 s
   "KM3" : Bool = PLC KM3 AT %Q2.2, 1 s
   "主电机启动JW1" : Bool = PLC 变频器上电 AT %Q2.3, 1 s
   "气垫调整防粘连KM19" : Bool = PLC 气垫调整防粘连KM19 AT %Q2.4, 1 s
   "润滑油泵启动KM11" : Bool = PLC 润滑油泵启动KM11 AT %Q2.7, 1 s
   "滑块调整防粘连KM5" : Bool = PLC 滑块调整防粘连KM5 AT %Q3.0, 1 s
   "制动器阀" : Bool = PLC 制动器阀 AT %Q12.7, 1 s
   "飞轮制动阀" : Bool = PLC 飞轮制动阀 AT %Q13.0, 1 s
   "下死点指示(1)" : Bool = PLC "下死点指示(1)" AT %Q10.0, 1 s
   "离合器阀" : Bool = PLC 离合器阀 AT %Q12.6, 1 s
   "平衡缸润滑阀" : Bool = PLC 平衡缸润滑阀 AT %Q12.5, 1 s
   "KA41主电机正转" : Bool = PLC KA41主电机正转 AT %Q3.3, 1 s
   "润滑油位低指示" : Bool = PLC 润滑油位低指示 AT %Q10.2, 1 s
   "润滑油位高指示" : Bool = PLC 润滑油位高指示 AT %Q10.3, 1 s
   "气垫润滑高压指示" : Bool = PLC 气垫润滑高压指示 AT %Q10.4, 1 s
   "润滑正常" : Bool = PLC 润滑正常 AT %M15.4, 1 s
   "过滤器正常" : Bool = PLC 过滤器正常 AT %M5.0, 1 s
   "140(1)" : Bool = PLC 140 AT %M201.5, 1 s

HMI tags "计数功能"
   "计数开关" : Bool = PLC 中继.计数开关, 1 s
   "产量到达(1)" : Bool = PLC 中继.产量到达 AT %DB1.DBX0.0, 1 s
   "当前产量(1)" : Int = PLC 中间变量.当前产量 AT %DB1.DBX0.0, 1 s
   "目标产量" : Int = PLC 中间变量.目标产量 AT %DB1.DBW0, 1 s
   "计数清零开关" : Bool = PLC 中继.计数清零开关 AT %DB1.DBW0, 1 s

discrete alarms
   1: '急停', class Errors, trigger "PLC报警变量组1" bit 0
   2: '润滑压力异常', class Errors, trigger "PLC报警变量组1" bit 1
   3: '"离合器压力异常', class Errors, trigger "PLC报警变量组1" bit 2
   4: '"平衡器压力异常"', class Errors, trigger "PLC报警变量组1" bit 3
   5: '"液压保护过载"', class Errors, trigger "PLC报警变量组1" bit 4
   6: '"低液位"', class Errors, trigger "PLC报警变量组1" bit 5
   7: '"滑块调整上限位断开"', class Errors, trigger "PLC报警变量组1" bit 6
   8: '"滑块调整下限位断开"', class Errors, trigger "PLC报警变量组1" bit 7
   9: '"双阀粘连1-K3"', class Errors, trigger "PLC报警变量组1" bit 8
   10: '"双阀粘连1-K4"', class Errors, trigger "PLC报警变量组1" bit 9
   11: '"双阀继电器粘连1"', class Errors, trigger "PLC报警变量组1" bit 10
   12: '"双阀继电器粘连2"', class Errors, trigger "PLC报警变量组1" bit 11
   13: '"润滑电机过载"', class Errors, trigger "PLC报警变量组1" bit 12
   14: '"工作台油泵电机过载"', class Errors, trigger "PLC报警变量组1" bit 13
   15: '"主电机过载"', class Errors, trigger "PLC报警变量组1" bit 14
   16: '"润滑异常"', class Errors, trigger "PLC报警变量组1" bit 15
   17: '工作台未夹紧', class Errors, trigger "PLC报警变量组2" bit 0
   18: '"工作台未眠放松"', class Errors, trigger "PLC报警变量组2" bit 1
   19: '"液压保护压力未正常"', class Errors, trigger "PLC报警变量组2" bit 2
   20: '"滑块调整电机过载"', class Errors, trigger "PLC报警变量组2" bit 3
   21: '"超载指示"', class Errors, trigger "PLC报警变量组2" bit 4
   22: '"气压未正常"', class Errors, trigger "PLC报警变量组2" bit 5
   23: '"急停中', class Errors, trigger "PLC报警变量组2" bit 6
   24: '异常报警', class Errors, trigger "PLC报警变量组2" bit 7
   25: '右前工作台未落下到位', class Errors, trigger "PLC报警变量组2" bit 8
   26: '左后工作台未落下到位', class Errors, trigger "PLC报警变量组2" bit 9
   27: '"右前工作台未顶起到位"', class Errors, trigger "PLC报警变量组2" bit 10
   28: '"左前工作台未顶起到位"', class Errors, trigger "PLC报警变量组2" bit 11
   29: '"工作台未开进到位"', class Errors, trigger "PLC报警变量组2" bit 12
   30: '左气垫未落下到位', class Errors, trigger "PLC报警变量组2" bit 13
   31: '中气垫未落下到位', class Errors, trigger "PLC报警变量组2" bit 14
   32: '右气垫未落下到位', class Errors, trigger "PLC报警变量组2" bit 15

screen "滑块角度" 800x480
   Circle "圆_2" at 245,51 size 21x21
      Appearance <- "360"
   Circle "圆_3" at 274,56 size 21x21
      Appearance <- "10度"
   Circle "圆_4" at 303,66 size 21x21
      Appearance <- "20度"
   Circle "圆_5" at 326,79 size 21x21
      Appearance <- "30度"
   Circle "圆_6" at 346,95 size 21x21
      Appearance <- "40度"
   Circle "圆_7" at 364,115 size 21x21
      Appearance <- "50"
   Circle "圆_8" at 377,135 size 21x21
      Appearance <- "60"
   Circle "圆_9" at 385,157 size 21x21
      Appearance <- "70"
   Circle "圆_10" at 392,179 size 21x21
      Appearance <- "80"
   Circle "圆_11" at 394,202 size 21x21
      Appearance <- "90"
   Circle "圆_12" at 391,226 size 21x21
      Appearance <- "100"
   Circle "圆_13" at 386,249 size 21x21
      Appearance <- "110"
   Circle "圆_14" at 378,271 size 21x21
      Appearance <- "120"
   Circle "圆_15" at 365,292 size 21x21
      Appearance <- "130"
   Circle "圆_16" at 348,311 size 21x21
      Appearance <- "140(1)"
   Circle "圆_17" at 328,328 size 21x21
      Appearance <- "150"
   Circle "圆_18" at 306,342 size 21x21
      Appearance <- "160"
   Circle "圆_19" at 276,353 size 21x21
      Appearance <- "170"
   Circle "圆_20" at 247,357 size 21x21
      Appearance <- "180"
   Circle "圆_22" at 219,352 size 21x21
      Appearance <- "190"
   Circle "圆_23" at 195,344 size 21x21
      Appearance <- "200"
   Circle "圆_24" at 172,333 size 21x21
      Appearance <- "210"
   Circle "圆_25" at 152,319 size 21x21
      Appearance <- "220"
   Circle "圆_26" at 133,302 size 21x21
      Appearance <- "230"
   Circle "圆_27" at 117,281 size 21x21
      Appearance <- "240"
   Circle "圆_28" at 104,258 size 21x21
      Appearance <- "250"
   Circle "圆_29" at 96,229 size 21x21
      Appearance <- "260"
   Circle "圆_30" at 93,201 size 21x21
      Appearance <- "270"
   Circle "圆_32" at 95,178 size 21x21
      Appearance <- "280"
   Circle "圆_33" at 100,155 size 21x21
      Appearance <- "290"
   Circle "圆_34" at 110,131 size 21x21
      Appearance <- "300"
   Circle "圆_35" at 126,111 size 21x21
      Appearance <- "310"
   Circle "圆_36" at 144,91 size 21x21
      Appearance <- "320"
   Circle "圆_37" at 167,74 size 21x21
      Appearance <- "330"
   Circle "圆_38" at 191,63 size 21x21
      Appearance <- "340"
   Circle "圆_39" at 218,54 size 21x21
      Appearance <- "350"
   TextField "文本域_2" at 422,193 size 43x40; Text '90'
   TextField "文本域_3" at 221,378 size 62x40; Text '180'
   TextField "文本域_5" at 196,183 size 117x31; Text '滑块位置'
   TextField "文本域_4" at 25,203 size 62x40; Text '270'
   TextField "文本域_1" at 241,12 size 24x40; Text '0'
   SymbolLibrary "符号库_1" at 515,6 size 138x90
   SymbolLibrary "符号库_2" at 680,47 size 86x40
   TextField "文本域_7" at 671,101 size 77x21; Text '滑块电机'
   TextField "文本域_6" at 562,103 size 59x21; Text '主电机'
   Circle "圆_21" at 687,27 size 14x14
      Appearance <- "滑块向上KM6"
   Circle "圆_31" at 729,27 size 14x14
      Appearance <- "滑块向下KM7"
   TextField "文本域_15" at 677,7 size 33x17; Text '向上'
   TextField "文本域_16" at 719,8 size 33x17; Text '向下'
   Button "按钮_1" at 28,424 size 67x56; TextOff '滑块角度'
      on Click: ActivateScreen("滑块角度", 0)
   Button "按钮_2" at 96,424 size 67x56; TextOff '设备状态'
      on Click: ActivateScreen("设备状态", 0)
   Button "按钮_3" at 163,424 size 71x55; TextOff '工作台操作'
      on Click: ActivateScreen("工作台操作", 0)
   Button "按钮_4" at 235,424 size 69x56; TextOff '气垫操作'
      on Click: ActivateScreen("气垫操作", 0)
   Button "按钮_5" at 304,423 size 66x57; TextOff '故障显示'
      on Click: ActivateScreen("故障显示", 0)
   Button "按钮_6" at 371,423 size 73x57; TextOff '输出显示'
      on Click: ActivateScreen("输出显示", 0)
   Button "按钮_7" at 445,422 size 66x58; TextOff '输入显示'
      on Click: ActivateScreen("输入显示", 0)
   IOField "I/O 域_1" at 228,217 size 56x32; FormatPattern 999
      ProcessValue <- "横梁编码器 _DB_+0.6"
   Button "按钮_8" at 514,423 size 68x56; TextOn '滑块调整'; TextOff '滑块调整'
      on Click: ActivateScreen("滑块调整", 0)
   Button "按钮_9" at 584,422 size 65x58; TextOff '报警信息'
      on Click: ActivateScreen("报警信息", 0)
   TextField "文本域_10" at 475,199 size 93x25; Text '当前产量'
   TextField "文本域_11" at 475,133 size 93x25; Text '设置产量'
   TextField "文本域_12" at 701,133 size 93x25; Text '计数清零'
   TextField "文本域_13" at 594,132 size 93x25; Text '计数通断'
   IOField "I/O 域_2" at 486,159 size 81x29; FormatPattern 9999
      ProcessValue <- "目标产量"
   IOField "I/O 域_3" at 486,225 size 87x32; FormatPattern 9999
      ProcessValue <- "当前产量(1)"
   Rectangle "矩形_1" at 487,264 size 88x60
      Appearance <- "产量到达"
      Visibility <- "产量到达(1)"
   TextField "文本域_14" at 486,283 size 85x23; Text '产量完成'
   Switch "开关_1" at 587,176 size 102x93; TextOn '通'; CaptionText 'Switch'; TextOff '断'
      Appearance <- "计数开始"
      ProcessValue <- "计数开关"
   Button "按钮_11" at 710,193 size 75x72; TextOff '清零'
      on Press: SetBit("计数清零开关")
      on Release: ResetBit("计数清零开关")
   TextField "文本域_17" at 391,344 size 93x25; Text '润滑故障'
   TextField "文本域_19" at 601,344 size 93x25; Text '平衡气压'
   TextField "文本域_20" at 698,344 size 93x25; Text '液压保护'
   TextField "文本域_21" at 499,345 size 93x25; Text '离制压力'
   Circle "圆_42" at 234,95 size 47x47
      Appearance <- "上死点"
   TextField "文本域_8" at 234,110 size 47x17; Text '上死点'
   Circle "圆_43" at 235,290 size 47x47
      Appearance <- "下死点"
   TextField "文本域_9" at 236,305 size 47x17; Text '下死点'
   Circle "圆_44" at 423,380 size 32x32
      Appearance <- "润滑正常"
   Circle "圆_48" at 48,19 size 56x56
      Appearance <- "润滑油泵启动OK"
   TextField "文本域_18" at 27,74 size 89x17; Text '润滑电机运行'
   Circle "圆_49" at 546,20 size 56x56
      Appearance <- "主电机运行指示"

screen "设备状态" 800x480
   TextField "文本域_1" at 63,79 size 101x27; Text '润滑正常'
   TextField "文本域_2" at 64,142 size 101x27; Text '急停正常'
   TextField "文本域_3" at 50,205 size 125x27; Text '工作台夹紧'
   TextField "文本域_4" at 66,268 size 101x27; Text '气压正常'
   TextField "文本域_5" at 46,331 size 149x27; Text '液压保护正常'
   Circle "圆_1" at 325,208 size 27x27
      Appearance <- "工作台落到位前(1)"
   TextField "文本域_6" at 293,237 size 96x16; Text '工作台前落到位'
   Circle "圆_2" at 427,207 size 27x27
      Appearance <- "工作台落到位后(1)"
   TextField "文本域_7" at 395,237 size 96x16; Text '工作台后落到位'
   Circle "圆_3" at 527,207 size 27x27
      Appearance <- "工作台夹紧压检"
   TextField "文本域_8" at 495,237 size 96x16; Text '工作台夹紧压力'
   Circle "圆_4" at 223,207 size 27x27
      Appearance <- "工作台夹紧阀(1)"
   TextField "文本域_9" at 198,237 size 83x16; Text '工作台夹紧阀'
   Circle "圆_5" at 427,81 size 27x27
      Appearance <- "润滑油压正常"
   TextField "文本域_10" at 399,111 size 83x16; Text '润滑油压正常'
   Circle "圆_7" at 325,81 size 27x27
      Appearance <- "过滤器正常"
   TextField "文本域_12" at 295,111 size 96x16; Text '润滑过滤器正常'
   Circle "圆_8" at 222,81 size 27x27
      Appearance <- "工作台落到位后"
   TextField "文本域_13" at 196,111 size 83x16; Text '润滑油位正常'
   Circle "圆_9" at 527,81 size 27x27
      Appearance <- "工作台落到位后"
   TextField "文本域_14" at 502,111 size 83x16; Text '润滑频次正常'
   Circle "圆_10" at 325,270 size 27x27
      Appearance <- "工作台落到位前"
   TextField "文本域_15" at 306,299 size 70x16; Text '离合器压力'
   Circle "圆_11" at 427,269 size 27x27
      Appearance <- "工作台落到位后"
   Circle "圆_12" at 223,269 size 27x27
      Appearance <- "平衡缸气压检测"
   TextField "文本域_16" at 200,298 size 70x16; Text '平衡缸压力'
   TextField "文本域_17" at 407,300 size 70x16; Text '制动器压力'
   Circle "圆_6" at 615,81 size 27x27
      Appearance <- "润滑油泵启动OK"
   TextField "文本域_11" at 590,111 size 83x16; Text '润滑电机启动'
   Circle "圆_14" at 325,141 size 27x27
      Appearance <- "急停开点2"
   TextField "文本域_19" at 312,171 size 71x16; Text '急停开点2#'
   Circle "圆_15" at 222,141 size 27x27
      Appearance <- "急停开点1"
   TextField "文本域_20" at 207,171 size 71x16; Text '急停开点1#'
   Circle "圆_16" at 527,142 size 27x27
      Appearance <- "爬梯开关"
   TextField "文本域_21" at 511,171 size 57x16; Text '梯子开关'
   Circle "圆_18" at 325,333 size 27x27
      Appearance <- "液压保护卸荷"
   TextField "文本域_23" at 306,362 size 70x16; Text '卸荷阀卸荷'
   Circle "圆_19" at 427,332 size 27x27
      Appearance <- "液压保护故障"
   Circle "圆_20" at 223,332 size 27x27
      Appearance <- "液压保护压力检测"
   TextField "文本域_24" at 200,361 size 83x16; Text '液压保护压力'
   TextField "文本域_25" at 407,363 size 57x16; Text '系统压力'
   Button "按钮_1" at 28,424 size 67x56; TextOn '滑块角度'; TextOff '滑块角度'
      on Click: ActivateScreen("滑块角度", 0)
   Button "按钮_2" at 96,424 size 67x56; TextOn '设备状态'; TextOff '设备状态'
      on Click: ActivateScreen("设备状态", 0)
   Button "按钮_3" at 163,424 size 71x55; TextOn '工作台操作'; TextOff '工作台操作'
      on Click: ActivateScreen("工作台操作", 0)
   Button "按钮_4" at 235,424 size 69x56; TextOn '气垫操作'; TextOff '气垫操作'
      on Click: ActivateScreen("气垫操作", 0)
   Button "按钮_5" at 304,423 size 66x57; TextOn '故障显示'; TextOff '故障显示'
      on Click: ActivateScreen("故障显示", 0)
   Button "按钮_6" at 371,423 size 73x57; TextOn '输出显示'; TextOff '输出显示'
      on Click: ActivateScreen("输出显示", 0)
   Button "按钮_7" at 445,422 size 66x58; TextOn '输入显示'; TextOff '输入显示'
      on Click: ActivateScreen("输入显示", 0)
   Button "按钮_8" at 514,423 size 68x56; TextOn '滑块调整'; TextOff '滑块调整'
      on Click: ActivateScreen("滑块调整", 0)
   Button "按钮_9" at 592,422 size 65x58; TextOn '报警信息'; TextOff '报警信息'
      on Click: ActivateScreen("报警信息", 0)
   Circle "圆_13" at 427,144 size 27x27
      Appearance <- "急停闭点"
   TextField "文本域_18" at 412,171 size 71x16; Text '急停闭点2#'

